(* IEC 61131-3 sources: TAuto/IEC 61131-3, 10 files *)

(* ---- FB_MB_PULL v.3.st ---- *)
FUNCTION_BLOCK MB_PULL

(* MB_PULL v.3 *)

(* MB_PULL - функциональный блок опроса по протоколу Modbus *)

(* Внешне задаются такие параметры как:
   - Команда выполнения/остановки цикла (ExecuteType);
   - Адрес/номер Slave-устройства (SlaveId);
   - Команда Modbus, которая реализована в FB MB_RTU_MASTER (Mode; 1, 2, 3, 4, 5, 6, 15, 16);
   - Начальный адрес регистров (Address);
   - Количество считываемых/записываемых данных (Count). *)
(* Внешне реализованы функции чтения/записи массива данных, в зависимости от  выбранной функции *)
(* Внутри функционального блока опроса используются следующие библиотечные функции:
   - MB_RTU_MASTER - функциональный блок Modbus;
   - MB_MASTER_QUEUE - структура созданная для команд Modbus. *)

// Первоначальная проверка, блок не выполняется
// MB_MS - экземпляр FB MB_RTU_MASTER
IF NOT MB_MS.Busy THEN                                                            // True - выполняется команда, False - не выполняется клманда

   QUEUE_INDEX := MB_Q.CurrentCommandIndex;                                       // Тип QUEUE_INDEX - INT. MB_Q - экземпляр MB_MASTER_QUEUE

   // Текущая команда завершилась
   IF MB_MS.Done THEN                                                             // Признак того, что команда завершилась

      // Текущий индекс команды
      MB_Q.CurrentCommandIndex := MB_Q.CurrentCommandIndex + 1;

      // Нет ошибок при выполнении FB
      IF MB_MS.Error = 0 THEN                                                     // 1. 0 - ошибок нет. 2. Диапазон 1..1000 - ошибки устройства Modbus. 3. Диапазон 1000..2000 - ошибки СПО. 4. Диапазон 2000+ - ошибки блока MB_RTU_MASTER

         // Задан корреткный режим выполнения
         IF  MB_Q.Commands[QUEUE_INDEX].ExecuteType <> 0 THEN

            // Сброс флага для режима "одиночного выполнения"
            IF MB_Q.Commands[QUEUE_INDEX].ExecuteType = 255 THEN

               MB_Q.Commands[QUEUE_INDEX].ExecuteType := 0;

            END_IF;

            (* Закомментированно потому что реализовано во внешних ST-программах *)

            // // Для операций чтения данных (1, 2, 3, 4 функции Modbus)
            // IF MB_Q.Commands[QUEUE_INDEX].Mode = 1                                // Чтение значений из нескольких регистров флагов - Read Coil Status
            //   OR MB_Q.Commands[QUEUE_INDEX].Mode = 2                              // Чтение значений из нескольких дискретных входов - Read Discrete Inputs
            //   OR MB_Q.Commands[QUEUE_INDEX].Mode = 3                              // Чтение значений из нескольких регистров хранения - Read Holding Registers
            //   OR MB_Q.Commands[QUEUE_INDEX].Mode = 4 THEN                         // Чтение значений из нескольких регистров ввода - Read Input Registers

            //   // Копирование данных полученных с устройства
            //   MB_Q.Commands[QUEUE_INDEX].Data := MB_MS.DataOut;                   // Массив считанных данных из Slave-устройства

            // END_IF;
         END_IF;
      END_IF;
   END_IF;

   // Сброс индекса запросов
   IF QUEUE_INDEX = 49 THEN

      MB_Q.CurrentCommandIndex := 0;

   END_IF;

   // Циклический перебор "карты памяти"
   FOR COMMAND_INDEX := MB_Q.CurrentCommandIndex TO 49 DO                            // Тип COMMAND_INDEX - INT

      // Сохранение текущего индекса
      MB_Q.CurrentCommandIndex := COMMAND_INDEX;

      // Задан корреткный режим выполнения
      IF MB_Q.Commands[COMMAND_INDEX].ExecuteType <> 0 THEN

         // Режим "выполнить один раз"
         IF MB_Q.Commands[COMMAND_INDEX].ExecuteType = 2 THEN

            MB_Q.Commands[COMMAND_INDEX].ExecuteType := 255;

         END_IF;

         (* Закомментированно потому что реализовано во внешних ST-программах *)

         // // Для операций записи данных (5, 6, 15, 16 функции Modbus)
         // IF  MB_Q.Commands[COMMAND_INDEX].Mode = 5                                   // Запись значения одного флага - Force Single Coil
         //    OR MB_Q.Commands[COMMAND_INDEX].Mode = 6                                 // Запись значения в один регистр хранения - Preset Single Register
         //    OR MB_Q.Commands[COMMAND_INDEX].Mode = 15                                // Запись значений в несколько регистров флагов - Force Multiple Coils
         //    OR MB_Q.Commands[COMMAND_INDEX].Mode = 16 THEN                           // Запись значений в несколько регистров хранения - Preset Multiple Registers

         //    // Копирование данных для записи в устройство
         //    MB_MS.DataIn := MB_Q.Commands[COMMAND_INDEX].Data;                       // Массив данных для записи в Slave-устройство

         // END_IF;

         // Настрока FB MB_RTU_MASTER
         MB_MS.Request := MB_REQUEST;                                                // Тип MB_REQUEST - BOOL. Команда выполнения/остановки опроса. Срабатывает по фронту, т.е. при смене входа с False на True
         MB_MS.SlaveId := MB_Q.Commands[COMMAND_INDEX].SlaveId;                      // Адрес/номер Slave-устройства
         MB_MS.Mode := MB_Q.Commands[COMMAND_INDEX].Mode;                            // Команда Modbus (1, 2, 3, 4, 5, 6, 15, 16)
         MB_MS.Address := MB_Q.Commands[COMMAND_INDEX].Address;                      // Начальный адрес register/coil (0 - 65535)
         MB_MS.Count := MB_Q.Commands[COMMAND_INDEX].Count;                          // Количество считываемых/записываемых данных. Зависит от типа данных register/coil (0 -123 для регистров , 0-246 для бит)

         EXIT;
      END_IF;
   END_FOR;
END_IF;

// Настройка параметров обмена FB MB_RTU_MASTER
MB_MS.BaudRate := MB_BaudRate;                                                       // Тип MB_BaudRate - UDINT. Скорость (9600, 19200, 38400, 57600, 115200 и др.)
MB_MS.Parity := MB_Parity;                                                           // Тип MB_Parity - BOOL. Бит чётности (True - есть контроль чётности)
MB_MS.StopBit := MB_StopBit;                                                         // Тип MB_StopBit - USINT. Количество стоповых бит (1, 2)
MB_MS.DataBit := MB_DataBit;                                                         // Тип MB_DataBit - USINT. Количество бит данных (7, 8)
MB_MS.TimeOut := MB_TimeOut;                                                         // Тип MB_TimeOut - UDINT. Время ожидания выполнения команды, мс
MB_MS.BusNumber := MB_BusNumber;                                                     // Тип MB_BusNumber - USINT. Локальная шина БЦП - 0,1; TCM/MI01 - 2-99
MB_MS.PortNumber := MB_PortNumber;                                                   // Тип MB_PortNumber - USINT. Номер порта/канала (0, 1. Если используется ТСМ, то значения: 0-7)
MB_MS();                                                                             // Вызов блока MB_RTUMASTER

// Вывод информации из блока MB_RTU_MASTER
// MB_DataOut := MB_MS.DataOut;                                                      // Тип MB_DataOut - USINT_0_245. Результаты выполнения опроса
MB_Busy := MB_MS.Busy;                                                            // Тип MB_Busy - BOOL. Выставляется в true если выполняется команда
MB_Done := MB_MS.Done;                                                            // Тип MB_Done - BOOL. Признак того, что команда завершилась
MB_Error := MB_MS.Error;                                                          // Тип MB_Error - UDINT. Ошибка
MB_ExecutionTime := MB_MS.ExecutionTime;                                          // Тип MB_ExecutionTime - UDINT. Время выполнения последней команды, мс
MB_AverageExecutionTime := MB_MS.AverageExecutionTime;                            // Тип MB_AverageExecutionTime - UDINT. Время выполнения последних четырёх команд, мс

// Сброс команды выполнения
// Закоментировать без вызова блока MB_RTUMASTER
IF MB_MS.Request THEN                                                             // Команда выполнения/остановки опроса. Срабатывает по фронту, т.е. при смене входа с False на True

   MB_MS.Request := False;                                                        // Остановка команды выполнения опроса

END_IF;

END_FUNCTION_BLOCK

(* ---- FB_MB_PULL v.4.st ---- *)
FUNCTION_BLOCK MB_PULL

(* MB_PULL v.3 *)

(* MB_PULL - функциональный блок опроса по протоколу Modbus *)

(* Внешне задаются такие параметры как:
   - Команда выполнения/остановки цикла (ExecuteType);
   - Адрес/номер Slave-устройства (SlaveId);
   - Команда Modbus, которая реализована в FB MB_RTU_MASTER (Mode; 1, 2, 3, 4, 5, 6, 15, 16);
   - Начальный адрес регистров (Address);
   - Количество считываемых/записываемых данных (Count). *)
(* Внешне реализованы функции чтения/записи массива данных, в зависимости от  выбранной функции *)
(* Внутри функционального блока опроса используются следующие библиотечные функции:
   - MB_RTU_MASTER - функциональный блок Modbus;
   - MB_MASTER_QUEUE - структура созданная для команд Modbus. *)

// Первоначальная проверка, блок не выполняется
// MB_MS - экземпляр FB MB_RTU_MASTER

HV_1185557(.Request, .SlaveId, .TimeOut, .Mode, .Address, .DataIn, .Count);
            BOOL       USINT     UDINT    USINT   UINT  USINT_0_245  UINT

  .DataOut, .Busy, .Done, .Error, .ExecutionTime, .AverageExecutionTime
 USINT_0_245  BOOL  BOOL   UDINT    UDINT             UDINT

MB_COM (ExecuteType, SlaveId, Mode, Address, Count)
        USINT           USINT  USINT UINT   UINT

MB_QUEUE(Commands, CurrentCommandIndex)
            [0..49]
        MB_COM_0_49        INT

IF NOT MB_MS.Busy THEN                                                            // True - выполняется команда, False - не выполняется клманда

   QUEUE_INDEX := MB_Q.CurrentCommandIndex;                                       // Тип QUEUE_INDEX - INT. MB_Q - экземпляр MB_MASTER_QUEUE

   // Текущая команда завершилась
   IF MB_MS.Done THEN                                                             // Признак того, что команда завершилась

      // Текущий индекс команды
      MB_Q.CurrentCommandIndex := MB_Q.CurrentCommandIndex + 1;

      // Нет ошибок при выполнении FB
      IF MB_MS.Error = 0 THEN                                                     // 1. 0 - ошибок нет. 2. Диапазон 1..1000 - ошибки устройства Modbus. 3. Диапазон 1000..2000 - ошибки СПО. 4. Диапазон 2000+ - ошибки блока MB_RTU_MASTER

         // Задан корреткный режим выполнения
         IF  MB_Q.Commands[QUEUE_INDEX].ExecuteType <> 0 THEN

            // Сброс флага для режима "одиночного выполнения"
            IF MB_Q.Commands[QUEUE_INDEX].ExecuteType = 255 THEN

               MB_Q.Commands[QUEUE_INDEX].ExecuteType := 0;

            END_IF;

            (* Закомментированно потому что реализовано во внешних ST-программах *)

            // // Для операций чтения данных (1, 2, 3, 4 функции Modbus)
            // IF MB_Q.Commands[QUEUE_INDEX].Mode = 1                                // Чтение значений из нескольких регистров флагов - Read Coil Status
            //   OR MB_Q.Commands[QUEUE_INDEX].Mode = 2                              // Чтение значений из нескольких дискретных входов - Read Discrete Inputs
            //   OR MB_Q.Commands[QUEUE_INDEX].Mode = 3                              // Чтение значений из нескольких регистров хранения - Read Holding Registers
            //   OR MB_Q.Commands[QUEUE_INDEX].Mode = 4 THEN                         // Чтение значений из нескольких регистров ввода - Read Input Registers

            //   // Копирование данных полученных с устройства
            //   MB_Q.Commands[QUEUE_INDEX].Data := MB_MS.DataOut;                   // Массив считанных данных из Slave-устройства

            // END_IF;
         END_IF;
      END_IF;
   END_IF;

   // Сброс индекса запросов
   IF QUEUE_INDEX = 49 THEN

      MB_Q.CurrentCommandIndex := 0;

   END_IF;

   // Циклический перебор "карты памяти"
   FOR COMMAND_INDEX := MB_Q.CurrentCommandIndex TO 49 DO                            // Тип COMMAND_INDEX - INT

      // Сохранение текущего индекса
      MB_Q.CurrentCommandIndex := COMMAND_INDEX;

      // Задан корреткный режим выполнения
      IF MB_Q.Commands[COMMAND_INDEX].ExecuteType <> 0 THEN

         // Режим "выполнить один раз"
         IF MB_Q.Commands[COMMAND_INDEX].ExecuteType = 2 THEN

            MB_Q.Commands[COMMAND_INDEX].ExecuteType := 255;

         END_IF;

         (* Закомментированно потому что реализовано во внешних ST-программах *)

         // // Для операций записи данных (5, 6, 15, 16 функции Modbus)
         // IF  MB_Q.Commands[COMMAND_INDEX].Mode = 5                                   // Запись значения одного флага - Force Single Coil
         //    OR MB_Q.Commands[COMMAND_INDEX].Mode = 6                                 // Запись значения в один регистр хранения - Preset Single Register
         //    OR MB_Q.Commands[COMMAND_INDEX].Mode = 15                                // Запись значений в несколько регистров флагов - Force Multiple Coils
         //    OR MB_Q.Commands[COMMAND_INDEX].Mode = 16 THEN                           // Запись значений в несколько регистров хранения - Preset Multiple Registers

         //    // Копирование данных для записи в устройство
         //    MB_MS.DataIn := MB_Q.Commands[COMMAND_INDEX].Data;                       // Массив данных для записи в Slave-устройство

         // END_IF;

         // Настрока FB MB_RTU_MASTER
         MB_MS.Request := MB_REQUEST;                                                // Тип MB_REQUEST - BOOL. Команда выполнения/остановки опроса. Срабатывает по фронту, т.е. при смене входа с False на True
         MB_MS.SlaveId := MB_Q.Commands[COMMAND_INDEX].SlaveId;                      // Адрес/номер Slave-устройства
         MB_MS.Mode := MB_Q.Commands[COMMAND_INDEX].Mode;                            // Команда Modbus (1, 2, 3, 4, 5, 6, 15, 16)
         MB_MS.Address := MB_Q.Commands[COMMAND_INDEX].Address;                      // Начальный адрес register/coil (0 - 65535)
         MB_MS.Count := MB_Q.Commands[COMMAND_INDEX].Count;                          // Количество считываемых/записываемых данных. Зависит от типа данных register/coil (0 -123 для регистров , 0-246 для бит)

         EXIT;
      END_IF;
   END_FOR;
END_IF;

// Настройка параметров обмена FB MB_RTU_MASTER
MB_MS.BaudRate := MB_BaudRate;                                                       // Тип MB_BaudRate - UDINT. Скорость (9600, 19200, 38400, 57600, 115200 и др.)
MB_MS.Parity := MB_Parity;                                                           // Тип MB_Parity - BOOL. Бит чётности (True - есть контроль чётности)
MB_MS.StopBit := MB_StopBit;                                                         // Тип MB_StopBit - USINT. Количество стоповых бит (1, 2)
MB_MS.DataBit := MB_DataBit;                                                         // Тип MB_DataBit - USINT. Количество бит данных (7, 8)
MB_MS.TimeOut := MB_TimeOut;                                                         // Тип MB_TimeOut - UDINT. Время ожидания выполнения команды, мс
MB_MS.BusNumber := MB_BusNumber;                                                     // Тип MB_BusNumber - USINT. Локальная шина БЦП - 0,1; TCM/MI01 - 2-99
MB_MS.PortNumber := MB_PortNumber;                                                   // Тип MB_PortNumber - USINT. Номер порта/канала (0, 1. Если используется ТСМ, то значения: 0-7)
MB_MS();                                                                             // Вызов блока MB_RTUMASTER

// Вывод информации из блока MB_RTU_MASTER
// MB_DataOut := MB_MS.DataOut;                                                      // Тип MB_DataOut - USINT_0_245. Результаты выполнения опроса
MB_Busy := MB_MS.Busy;                                                            // Тип MB_Busy - BOOL. Выставляется в true если выполняется команда
MB_Done := MB_MS.Done;                                                            // Тип MB_Done - BOOL. Признак того, что команда завершилась
MB_Error := MB_MS.Error;                                                          // Тип MB_Error - UDINT. Ошибка
MB_ExecutionTime := MB_MS.ExecutionTime;                                          // Тип MB_ExecutionTime - UDINT. Время выполнения последней команды, мс
MB_AverageExecutionTime := MB_MS.AverageExecutionTime;                            // Тип MB_AverageExecutionTime - UDINT. Время выполнения последних четырёх команд, мс

// Сброс команды выполнения
// Закоментировать без вызова блока MB_RTUMASTER
IF MB_MS.Request THEN                                                             // Команда выполнения/остановки опроса. Срабатывает по фронту, т.е. при смене входа с False на True

   MB_MS.Request := False;                                                        // Остановка команды выполнения опроса

END_IF;

END_FUNCTION_BLOCK

(* ---- FUNCTION_BLOCK MB_PULL.st ---- *)
FUNCTION_BLOCK MB_PULL

(* MB_PULL v.3 *)

(* MB_PULL - функциональный блок опроса по протоколу Modbus *)

(* Внешне задаются такие параметры как:
   - Команда выполнения/остановки цикла (ExecuteType);
   - Адрес/номер Slave-устройства (SlaveId);
   - Команда Modbus, которая реализована в FB MB_RTU_MASTER (Mode; 1, 2, 3, 4, 5, 6, 15, 16);
   - Начальный адрес регистров (Address);
   - Количество считываемых/записываемых данных (Count). *)
(* Внешне реализованы функции чтения/записи массива данных, в зависимости от  выбранной функции *)
(* Внутри функционального блока опроса используются следующие библиотечные функции:
   - MB_RTU_MASTER - функциональный блок Modbus;
   - MB_MASTER_QUEUE - структура созданная для команд Modbus. *)

// Первоначальная проверка, блок не выполняется
// MB_MS - экземпляр FB MB_RTU_MASTER
IF NOT MB_MS.Busy THEN                                                            // True - выполняется команда, False - не выполняется клманда

    // Текущая команда завершилась
    IF MB_MS.Done THEN                                                             // Признак того, что команда завершилась

    // Текущий индекс команды
    MB_Q.CurrentCommandIndex := MB_Q.CurrentCommandIndex + 1;

        // Нет ошибок при выполнении FB
        IF MB_MS.Error = 0 THEN                                                     // 1. 0 - ошибок нет. 2. Диапазон 1..1000 - ошибки устройства Modbus. 3. Диапазон 1000..2000 - ошибки СПО. 4. Диапазон 2000+ - ошибки блока MB_RTU_MASTER

CASE MB_Q.CurrentCommandIndex OF
1:
QUEUE_INDEX := 1;
2:
QUEUE_INDEX := 2;
3:
QUEUE_INDEX := 3;
4:
QUEUE_INDEX := 4;
5:
QUEUE_INDEX := 5;
6:
QUEUE_INDEX := 6;
7:
QUEUE_INDEX := 7;
8:
QUEUE_INDEX := 8;
9:
QUEUE_INDEX := 9;
10:
QUEUE_INDEX := 10;
MB_Q.CurrentCommandIndex := 0;
END_CASE;

         // Задан корреткный режим выполнения
         IF  MB_Q.Commands[QUEUE_INDEX].ExecuteType <> 0 THEN

            // Сброс флага для режима "одиночного выполнения"
            IF MB_Q.Commands[QUEUE_INDEX].ExecuteType = 255 THEN

               MB_Q.Commands[QUEUE_INDEX].ExecuteType := 0;

            END_IF;

                    END_IF;
      END_IF;
   END_IF;

   // Сброс индекса запросов
   IF QUEUE_INDEX = 49 THEN

      MB_Q.CurrentCommandIndex := 0;

   END_IF;

   // Циклический перебор "карты памяти"
   FOR COMMAND_INDEX := MB_Q.CurrentCommandIndex TO 49 DO                            // Тип COMMAND_INDEX - INT

      // Сохранение текущего индекса
      MB_Q.CurrentCommandIndex := COMMAND_INDEX;

      // Задан корреткный режим выполнения
      IF MB_Q.Commands[COMMAND_INDEX].ExecuteType <> 0 THEN

         // Режим "выполнить один раз"
         IF MB_Q.Commands[COMMAND_INDEX].ExecuteType = 2 THEN

            MB_Q.Commands[COMMAND_INDEX].ExecuteType := 255;

         END_IF;

         (* Закомментированно потому что реализовано во внешних ST-программах *)

         // // Для операций записи данных (5, 6, 15, 16 функции Modbus)
         // IF  MB_Q.Commands[COMMAND_INDEX].Mode = 5                                   // Запись значения одного флага - Force Single Coil
         //    OR MB_Q.Commands[COMMAND_INDEX].Mode = 6                                 // Запись значения в один регистр хранения - Preset Single Register
         //    OR MB_Q.Commands[COMMAND_INDEX].Mode = 15                                // Запись значений в несколько регистров флагов - Force Multiple Coils
         //    OR MB_Q.Commands[COMMAND_INDEX].Mode = 16 THEN                           // Запись значений в несколько регистров хранения - Preset Multiple Registers

         //    // Копирование данных для записи в устройство
         //    MB_MS.DataIn := MB_Q.Commands[COMMAND_INDEX].Data;                       // Массив данных для записи в Slave-устройство

         // END_IF;

         // Настрока FB MB_RTU_MASTER
         MB_MS.Request := MB_REQUEST;                                                // Тип MB_REQUEST - BOOL. Команда выполнения/остановки опроса. Срабатывает по фронту, т.е. при смене входа с False на True
         MB_MS.SlaveId := MB_Q.Commands[COMMAND_INDEX].SlaveId;                      // Адрес/номер Slave-устройства
         MB_MS.Mode := MB_Q.Commands[COMMAND_INDEX].Mode;                            // Команда Modbus (1, 2, 3, 4, 5, 6, 15, 16)
         MB_MS.Address := MB_Q.Commands[COMMAND_INDEX].Address;                      // Начальный адрес register/coil (0 - 65535)
         MB_MS.Count := MB_Q.Commands[COMMAND_INDEX].Count;                          // Количество считываемых/записываемых данных. Зависит от типа данных register/coil (0 -123 для регистров , 0-246 для бит)

         EXIT;
      END_IF;
   END_FOR;
END_IF;

// Настройка параметров обмена FB MB_RTU_MASTER
MB_MS.BaudRate := MB_BaudRate;                                                       // Тип MB_BaudRate - UDINT. Скорость (9600, 19200, 38400, 57600, 115200 и др.)
MB_MS.Parity := MB_Parity;                                                           // Тип MB_Parity - BOOL. Бит чётности (True - есть контроль чётности)
MB_MS.StopBit := MB_StopBit;                                                         // Тип MB_StopBit - USINT. Количество стоповых бит (1, 2)
MB_MS.DataBit := MB_DataBit;                                                         // Тип MB_DataBit - USINT. Количество бит данных (7, 8)
MB_MS.TimeOut := MB_TimeOut;                                                         // Тип MB_TimeOut - UDINT. Время ожидания выполнения команды, мс
MB_MS.BusNumber := MB_BusNumber;                                                     // Тип MB_BusNumber - USINT. Локальная шина БЦП - 0,1; TCM/MI01 - 2-99
MB_MS.PortNumber := MB_PortNumber;                                                   // Тип MB_PortNumber - USINT. Номер порта/канала (0, 1. Если используется ТСМ, то значения: 0-7)
MB_MS();                                                                             // Вызов блока MB_RTUMASTER

// Вывод информации из блока MB_RTU_MASTER
// MB_DataOut := MB_MS.DataOut;                                                      // Тип MB_DataOut - USINT_0_245. Результаты выполнения опроса
MB_Busy := MB_MS.Busy;                                                            // Тип MB_Busy - BOOL. Выставляется в true если выполняется команда
MB_Done := MB_MS.Done;                                                            // Тип MB_Done - BOOL. Признак того, что команда завершилась
MB_Error := MB_MS.Error;                                                          // Тип MB_Error - UDINT. Ошибка
MB_ExecutionTime := MB_MS.ExecutionTime;                                          // Тип MB_ExecutionTime - UDINT. Время выполнения последней команды, мс
MB_AverageExecutionTime := MB_MS.AverageExecutionTime;                            // Тип MB_AverageExecutionTime - UDINT. Время выполнения последних четырёх команд, мс

// Сброс команды выполнения
// Закоментировать без вызова блока MB_RTUMASTER
IF MB_MS.Request THEN                                                             // Команда выполнения/остановки опроса. Срабатывает по фронту, т.е. при смене входа с False на True

   MB_MS.Request := False;                                                        // Остановка команды выполнения опроса

END_IF;

END_FUNCTION_BLOCK

(* ---- IO_control.st ---- *)
PROGRAM IO_control

(***************************************************************************)
// ЛОКАЛЬНАЯ ШИНА 0
(***************************************************************************)

// [2] DO32
_IO_Q1_DO32_0_VAL.Measurement := UB_0_0_DO32_CH0_OUT;
_IO_Q1_DO32_1_VAL.Measurement := UB_0_0_DO32_CH1_OUT;
_IO_Q1_DO32_2_VAL.Measurement := UB_0_0_DO32_CH2_OUT;
_IO_Q1_DO32_3_VAL.Measurement := UB_0_0_DO32_CH3_OUT;
_IO_Q1_DO32_4_VAL.Measurement := UB_0_0_DO32_CH4_OUT;
_IO_Q1_DO32_5_VAL.Measurement := UB_0_0_DO32_CH5_OUT;
_IO_Q1_DO32_6_VAL.Measurement := UB_0_0_DO32_CH6_OUT;
_IO_Q1_DO32_7_VAL.Measurement := UB_0_0_DO32_CH7_OUT;
_IO_Q1_DO32_8_VAL.Measurement := UB_0_0_DO32_CH8_OUT;
_IO_Q1_DO32_9_VAL.Measurement := UB_0_0_DO32_CH9_OUT;
_IO_Q1_DO32_10_VAL.Measurement := UB_0_0_DO32_CH10_OUT;
_IO_Q1_DO32_11_VAL.Measurement := UB_0_0_DO32_CH11_OUT;
_IO_Q1_DO32_12_VAL.Measurement := UB_0_0_DO32_CH12_OUT;
_IO_Q1_DO32_13_VAL.Measurement := UB_0_0_DO32_CH13_OUT;
_IO_Q1_DO32_14_VAL.Measurement := UB_0_0_DO32_CH14_OUT;
_IO_Q1_DO32_15_VAL.Measurement := UB_0_0_DO32_CH15_OUT;
_IO_Q1_DO32_16_VAL.Measurement := UB_0_0_DO32_CH16_OUT;
_IO_Q1_DO32_17_VAL.Measurement := UB_0_0_DO32_CH17_OUT;
_IO_Q1_DO32_18_VAL.Measurement := UB_0_0_DO32_CH18_OUT;
_IO_Q1_DO32_19_VAL.Measurement := UB_0_0_DO32_CH19_OUT;
_IO_Q1_DO32_20_VAL.Measurement := UB_0_0_DO32_CH20_OUT;
_IO_Q1_DO32_21_VAL.Measurement := UB_0_0_DO32_CH21_OUT;
_IO_Q1_DO32_22_VAL.Measurement := UB_0_0_DO32_CH22_OUT;
_IO_Q1_DO32_23_VAL.Measurement := UB_0_0_DO32_CH23_OUT;
_IO_Q1_DO32_24_VAL.Measurement := UB_0_0_DO32_CH24_OUT;
_IO_Q1_DO32_25_VAL.Measurement := UB_0_0_DO32_CH25_OUT;
_IO_Q1_DO32_26_VAL.Measurement := UB_0_0_DO32_CH26_OUT;
_IO_Q1_DO32_27_VAL.Measurement := UB_0_0_DO32_CH27_OUT;
_IO_Q1_DO32_28_VAL.Measurement := UB_0_0_DO32_CH28_OUT;
_IO_Q1_DO32_29_VAL.Measurement := UB_0_0_DO32_CH29_OUT;
_IO_Q1_DO32_30_VAL.Measurement := UB_0_0_DO32_CH30_OUT;
_IO_Q1_DO32_31_VAL.Measurement := UB_0_0_DO32_CH31_OUT;

END_PROGRAM

(* ---- IO_RT.st ---- *)
PROGRAM IO_RT

//ВЫЗОВ ГЕНЕРАТОРОВ
GENERATOR(.StartGener, .PulseTime, .ResetCnt);
SIG_GEN_1(.RUN, .PERIOD, .MAXIMUM);

// НАСТРОЙКА ФБ AD
AD_VALID_DOWN := -100000;
AD_VALID_UP := 100000;
AD_IN0 := 10;
AD_IN100 := 100;

// КВИТИРОВАНИЕ
TIMER_REAL(FALSE, 0, 0, 10, T#20ms);

TMB_1_0_DI32_KVIT := TIMER_REAL.Out;
TMB_1_0_DO32_KVIT := TIMER_REAL.Out;
TMB_1_0_AIG16_KVIT := TIMER_REAL.Out;
TMB_1_0_AI8_KVIT := TIMER_REAL.Out;
TMB_1_0_AOC4_KVIT := TIMER_REAL.Out;

// ИНТЕГРАЛЬНЫЙ ПОАЗАТЕЛЬ ШИНЫ
IF TMB_1_0_DI32_INTEGRAL_VAL_QUALITY AND
    TMB_1_0_DO32_INTEGRAL_VAL_DIAG_QUALITY AND
    TMB_1_0_AIG16_INTEGRAL_VAL_QUALITY AND
    TMB_1_0_AI8_INTEGRAL_VAL_QUALITY AND
    TMB_1_0_AOC4_INTEGRAL_VAL_DIAG_QUALITY

    THEN TMB_1_0_TMB_QUALITY := TRUE;
    ELSE TMB_1_0_TMB_QUALITY := FALSE;
END_IF;

END_PROGRAM

(* ---- IO_SF.st ---- *)
PROGRAM IO

//ВЫЗОВ ГЕНЕРАТОРОВ
GENERATOR(.StartGener, .PulseTime, .ResetCnt);
SIG_GEN_1(.RUN, .PERIOD, .MAXIMUM);

// НАСТРОЙКА ФБ AD
AD_VALID_DOWN := -100000;
AD_VALID_UP := 100000;
AD_IN0 := 10;
AD_IN100 := 100;

// КВИТИРОВАНИЕ
TIMER_REAL(FALSE, 0, 0, 10, T#20ms);

UB_0_0_DI32_KVIT := TIMER_REAL.Out;
UB_0_0_DO32_KVIT := TIMER_REAL.Out;
UB_0_0_AIG16_KVIT := TIMER_REAL.Out;
UB_0_0_AI8_KVIT := TIMER_REAL.Out;
UB_0_0_AOC4_KVIT := TIMER_REAL.Out;

UB_0_32_DI32_KVIT := TIMER_REAL.Out;
UB_0_32_DO32_KVIT := TIMER_REAL.Out;
UB_0_32_AIG16_KVIT := TIMER_REAL.Out;
UB_0_32_AI8_KVIT := TIMER_REAL.Out;
UB_0_32_AOC4_KVIT := TIMER_REAL.Out;

UB_1_0_DI32_KVIT := TIMER_REAL.Out;
UB_1_0_DO32_KVIT := TIMER_REAL.Out;
UB_1_0_AIG16_KVIT := TIMER_REAL.Out;
UB_1_0_AI8_KVIT := TIMER_REAL.Out;
UB_1_0_AOC4_KVIT := TIMER_REAL.Out;

UB_12_0_DI32_KVIT := TIMER_REAL.Out;
UB_12_0_DO32_KVIT := TIMER_REAL.Out;
UB_12_0_AIG16_KVIT := TIMER_REAL.Out;
UB_12_0_AI8_KVIT := TIMER_REAL.Out;
UB_12_0_AOC4_KVIT := TIMER_REAL.Out;

UB_22_0_DI32_KVIT := TIMER_REAL.Out;
UB_22_0_DO32_KVIT := TIMER_REAL.Out;
UB_22_0_AIG16_KVIT := TIMER_REAL.Out;
UB_22_0_AI8_KVIT := TIMER_REAL.Out;
UB_22_0_AOC4_KVIT := TIMER_REAL.Out;

// ИНТЕГРАЛЬНЫЙ ПОАЗАТЕЛЬ ШИНЫ
IF UB_0_0_DI32_INTEGRAL_VAL_QUALITY AND
    UB_0_0_DO32_INTEGRAL_VAL_DIAG_QUALITY AND
    UB_0_0_AIG16_INTEGRAL_VAL_QUALITY AND
    UB_0_0_AI8_INTEGRAL_VAL_QUALITY AND
    UB_0_0_AOC4_INTEGRAL_VAL_DIAG_QUALITY

    THEN UB_0_0_UNITBAS_QUALITY := TRUE;
    ELSE UB_0_0_UNITBAS_QUALITY := FALSE;
END_IF;

IF UB_0_32_DI32_INTEGRAL_VAL_QUALITY AND
    UB_0_32_DO32_INTEGRAL_VAL_DIAG_QUALITY AND
    UB_0_32_AIG16_INTEGRAL_VAL_QUALITY AND
    UB_0_32_AI8_INTEGRAL_VAL_QUALITY AND
    UB_0_32_AOC4_INTEGRAL_VAL_DIAG_QUALITY

    THEN UB_0_32_UNITBAS_QUALITY := TRUE;
    ELSE UB_0_32_UNITBAS_QUALITY := FALSE;
END_IF;

IF UB_1_0_DI32_INTEGRAL_VAL_QUALITY AND
    UB_1_0_DO32_INTEGRAL_VAL_DIAG_QUALITY AND
    UB_1_0_AIG16_INTEGRAL_VAL_QUALITY AND
    UB_1_0_AI8_INTEGRAL_VAL_QUALITY AND
    UB_1_0_AOC4_INTEGRAL_VAL_DIAG_QUALITY

    THEN UB_1_0_UNITBAS_QUALITY := TRUE;
    ELSE UB_1_0_UNITBAS_QUALITY := FALSE;
END_IF;

IF UB_12_0_DI32_INTEGRAL_VAL_QUALITY AND
    UB_12_0_DO32_INTEGRAL_VAL_DIAG_QUALITY AND
    UB_12_0_AIG16_INTEGRAL_VAL_QUALITY AND
    UB_12_0_AI8_INTEGRAL_VAL_QUALITY AND
    UB_12_0_AOC4_INTEGRAL_VAL_DIAG_QUALITY

    THEN UB_12_0_UNITBAS_QUALITY := TRUE;
    ELSE UB_12_0_UNITBAS_QUALITY := FALSE;
END_IF;

IF UB_22_0_DI32_INTEGRAL_VAL_QUALITY AND
    UB_22_0_DO32_INTEGRAL_VAL_DIAG_QUALITY AND
    UB_22_0_AIG16_INTEGRAL_VAL_QUALITY AND
    UB_22_0_AI8_INTEGRAL_VAL_QUALITY AND
    UB_22_0_AOC4_INTEGRAL_VAL_DIAG_QUALITY

    THEN UB_22_0_UNITBAS_QUALITY := TRUE;
    ELSE UB_22_0_UNITBAS_QUALITY := FALSE;
END_IF;

END_PROGRAM

(* ---- PRG CPU715_Modbus.st ---- *)
PROGRAM CPU715_Modbus

(* Программа для передачи данных по протоколу Modbus *)

(* Генерация осуществляется с помощью ФБ MultiTypeGener *)
(* Диапазон регистров:
        для IR, HR:
            DINT - 32000...41999
            REAL - 42000...51999
            INT - 52000...61999
        для CL, DI:
            BOOL - 32000...41999 *)
(* Используемые каналы 0-97 для каждого типа данных *)

(* Считывание CL регистров *)
    // Переменные BOOL, регистры - 32000...41999
        _IO_QX5_1_0 := RESVAR_BOOL;
        _IO_QX5_1_1 := RESVAR_BOOL;
        _IO_QX5_1_2 := RESVAR_BOOL;
        _IO_QX5_1_3 := RESVAR_BOOL;
        _IO_QX5_1_4 := RESVAR_BOOL;
        _IO_QX5_1_5 := RESVAR_BOOL;
        _IO_QX5_1_6 := RESVAR_BOOL;
        _IO_QX5_1_7 := RESVAR_BOOL;
        _IO_QX5_1_8 := RESVAR_BOOL;
        _IO_QX5_1_9 := RESVAR_BOOL;
        _IO_QX5_1_10 := RESVAR_BOOL;
        _IO_QX5_1_11 := RESVAR_BOOL;
        _IO_QX5_1_12 := RESVAR_BOOL;
        _IO_QX5_1_13 := RESVAR_BOOL;

        _IO_QX5_1_14 := RESVAR_BOOL;
        _IO_QX5_1_15 := RESVAR_BOOL;
        _IO_QX5_1_16 := RESVAR_BOOL;
        _IO_QX5_1_17 := RESVAR_BOOL;
        _IO_QX5_1_18 := RESVAR_BOOL;
        _IO_QX5_1_19 := RESVAR_BOOL;
        _IO_QX5_1_20 := RESVAR_BOOL;
        _IO_QX5_1_21 := RESVAR_BOOL;
        _IO_QX5_1_22 := RESVAR_BOOL;
        _IO_QX5_1_23 := RESVAR_BOOL;
        _IO_QX5_1_24 := RESVAR_BOOL;
        _IO_QX5_1_25 := RESVAR_BOOL;
        _IO_QX5_1_26 := RESVAR_BOOL;
        _IO_QX5_1_27 := RESVAR_BOOL;

        _IO_QX5_1_28 := RESVAR_BOOL;
        _IO_QX5_1_29 := RESVAR_BOOL;
        _IO_QX5_1_30 := RESVAR_BOOL;
        _IO_QX5_1_31 := RESVAR_BOOL;
        _IO_QX5_1_32 := RESVAR_BOOL;
        _IO_QX5_1_33 := RESVAR_BOOL;
        _IO_QX5_1_34 := RESVAR_BOOL;
        _IO_QX5_1_35 := RESVAR_BOOL;
        _IO_QX5_1_36 := RESVAR_BOOL;
        _IO_QX5_1_37 := RESVAR_BOOL;
        _IO_QX5_1_38 := RESVAR_BOOL;
        _IO_QX5_1_39 := RESVAR_BOOL;
        _IO_QX5_1_40 := RESVAR_BOOL;
        _IO_QX5_1_41 := RESVAR_BOOL;

        _IO_QX5_1_42 := RESVAR_BOOL;
        _IO_QX5_1_43 := RESVAR_BOOL;
        _IO_QX5_1_44 := RESVAR_BOOL;
        _IO_QX5_1_45 := RESVAR_BOOL;
        _IO_QX5_1_46 := RESVAR_BOOL;
        _IO_QX5_1_47 := RESVAR_BOOL;
        _IO_QX5_1_48 := RESVAR_BOOL;
        _IO_QX5_1_49 := RESVAR_BOOL;
        _IO_QX5_1_50 := RESVAR_BOOL;
        _IO_QX5_1_51 := RESVAR_BOOL;
        _IO_QX5_1_52 := RESVAR_BOOL;
        _IO_QX5_1_53 := RESVAR_BOOL;
        _IO_QX5_1_54 := RESVAR_BOOL;
        _IO_QX5_1_55 := RESVAR_BOOL;

        _IO_QX5_1_56 := RESVAR_BOOL;
        _IO_QX5_1_57 := RESVAR_BOOL;
        _IO_QX5_1_58 := RESVAR_BOOL;
        _IO_QX5_1_59 := RESVAR_BOOL;
        _IO_QX5_1_60 := RESVAR_BOOL;
        _IO_QX5_1_61 := RESVAR_BOOL;
        _IO_QX5_1_62 := RESVAR_BOOL;
        _IO_QX5_1_63 := RESVAR_BOOL;
        _IO_QX5_1_64 := RESVAR_BOOL;
        _IO_QX5_1_65 := RESVAR_BOOL;
        _IO_QX5_1_66 := RESVAR_BOOL;
        _IO_QX5_1_67 := RESVAR_BOOL;
        _IO_QX5_1_68 := RESVAR_BOOL;
        _IO_QX5_1_69 := RESVAR_BOOL;

        _IO_QX5_1_70 := RESVAR_BOOL;
        _IO_QX5_1_71 := RESVAR_BOOL;
        _IO_QX5_1_72 := RESVAR_BOOL;
        _IO_QX5_1_73 := RESVAR_BOOL;
        _IO_QX5_1_74 := RESVAR_BOOL;
        _IO_QX5_1_75 := RESVAR_BOOL;
        _IO_QX5_1_76 := RESVAR_BOOL;
        _IO_QX5_1_77 := RESVAR_BOOL;
        _IO_QX5_1_78 := RESVAR_BOOL;
        _IO_QX5_1_79 := RESVAR_BOOL;
        _IO_QX5_1_80 := RESVAR_BOOL;
        _IO_QX5_1_81 := RESVAR_BOOL;
        _IO_QX5_1_82 := RESVAR_BOOL;
        _IO_QX5_1_83 := RESVAR_BOOL;

        _IO_QX5_1_84 := RESVAR_BOOL;
        _IO_QX5_1_85 := RESVAR_BOOL;
        _IO_QX5_1_86 := RESVAR_BOOL;
        _IO_QX5_1_87 := RESVAR_BOOL;
        _IO_QX5_1_88 := RESVAR_BOOL;
        _IO_QX5_1_89 := RESVAR_BOOL;
        _IO_QX5_1_90 := RESVAR_BOOL;
        _IO_QX5_1_91 := RESVAR_BOOL;
        _IO_QX5_1_92 := RESVAR_BOOL;
        _IO_QX5_1_93 := RESVAR_BOOL;
        _IO_QX5_1_94 := RESVAR_BOOL;
        _IO_QX5_1_95 := RESVAR_BOOL;
        _IO_QX5_1_96 := RESVAR_BOOL;
        _IO_QX5_1_97 := RESVAR_BOOL;

(* Считывание DI регистров *)
    // Переменные BOOL, регистры - 32000...41999
        _IO_QU7_0 := RESVAR_BOOL;
        _IO_QU7_1 := RESVAR_BOOL;
        _IO_QU7_2 := RESVAR_BOOL;
        _IO_QU7_3 := RESVAR_BOOL;
        _IO_QU7_4 := RESVAR_BOOL;
        _IO_QU7_5 := RESVAR_BOOL;
        _IO_QU7_6 := RESVAR_BOOL;
        _IO_QU7_7 := RESVAR_BOOL;
        _IO_QU7_8 := RESVAR_BOOL;
        _IO_QU7_9 := RESVAR_BOOL;
        _IO_QU7_10 := RESVAR_BOOL;
        _IO_QU7_11 := RESVAR_BOOL;
        _IO_QU7_12 := RESVAR_BOOL;
        _IO_QU7_13 := RESVAR_BOOL;

        _IO_QU7_14 := RESVAR_BOOL;
        _IO_QU7_15 := RESVAR_BOOL;
        _IO_QU7_16 := RESVAR_BOOL;
        _IO_QU7_17 := RESVAR_BOOL;
        _IO_QU7_18 := RESVAR_BOOL;
        _IO_QU7_19 := RESVAR_BOOL;
        _IO_QU7_20 := RESVAR_BOOL;
        _IO_QU7_21 := RESVAR_BOOL;
        _IO_QU7_22 := RESVAR_BOOL;
        _IO_QU7_23 := RESVAR_BOOL;
        _IO_QU7_24 := RESVAR_BOOL;
        _IO_QU7_25 := RESVAR_BOOL;
        _IO_QU7_26 := RESVAR_BOOL;
        _IO_QU7_27 := RESVAR_BOOL;

        _IO_QU7_28 := RESVAR_BOOL;
        _IO_QU7_29 := RESVAR_BOOL;
        _IO_QU7_30 := RESVAR_BOOL;
        _IO_QU7_31 := RESVAR_BOOL;
        _IO_QU7_32 := RESVAR_BOOL;
        _IO_QU7_33 := RESVAR_BOOL;
        _IO_QU7_34 := RESVAR_BOOL;
        _IO_QU7_35 := RESVAR_BOOL;
        _IO_QU7_36 := RESVAR_BOOL;
        _IO_QU7_37 := RESVAR_BOOL;
        _IO_QU7_38 := RESVAR_BOOL;
        _IO_QU7_39 := RESVAR_BOOL;
        _IO_QU7_40 := RESVAR_BOOL;
        _IO_QU7_41 := RESVAR_BOOL;

        _IO_QU7_42 := RESVAR_BOOL;
        _IO_QU7_43 := RESVAR_BOOL;
        _IO_QU7_44 := RESVAR_BOOL;
        _IO_QU7_45 := RESVAR_BOOL;
        _IO_QU7_46 := RESVAR_BOOL;
        _IO_QU7_47 := RESVAR_BOOL;
        _IO_QU7_48 := RESVAR_BOOL;
        _IO_QU7_49 := RESVAR_BOOL;
        _IO_QU7_50 := RESVAR_BOOL;
        _IO_QU7_51 := RESVAR_BOOL;
        _IO_QU7_52 := RESVAR_BOOL;
        _IO_QU7_53 := RESVAR_BOOL;
        _IO_QU7_54 := RESVAR_BOOL;
        _IO_QU7_55 := RESVAR_BOOL;

        _IO_QU7_56 := RESVAR_BOOL;
        _IO_QU7_57 := RESVAR_BOOL;
        _IO_QU7_58 := RESVAR_BOOL;
        _IO_QU7_59 := RESVAR_BOOL;
        _IO_QU7_60 := RESVAR_BOOL;
        _IO_QU7_61 := RESVAR_BOOL;
        _IO_QU7_62 := RESVAR_BOOL;
        _IO_QU7_63 := RESVAR_BOOL;
        _IO_QU7_64 := RESVAR_BOOL;
        _IO_QU7_65 := RESVAR_BOOL;
        _IO_QU7_66 := RESVAR_BOOL;
        _IO_QU7_67 := RESVAR_BOOL;
        _IO_QU7_68 := RESVAR_BOOL;
        _IO_QU7_69 := RESVAR_BOOL;

        _IO_QU7_70 := RESVAR_BOOL;
        _IO_QU7_71 := RESVAR_BOOL;
        _IO_QU7_72 := RESVAR_BOOL;
        _IO_QU7_73 := RESVAR_BOOL;
        _IO_QU7_74 := RESVAR_BOOL;
        _IO_QU7_75 := RESVAR_BOOL;
        _IO_QU7_76 := RESVAR_BOOL;
        _IO_QU7_77 := RESVAR_BOOL;
        _IO_QU7_78 := RESVAR_BOOL;
        _IO_QU7_79 := RESVAR_BOOL;
        _IO_QU7_80 := RESVAR_BOOL;
        _IO_QU7_81 := RESVAR_BOOL;
        _IO_QU7_82 := RESVAR_BOOL;
        _IO_QU7_83 := RESVAR_BOOL;

        _IO_QU7_84 := RESVAR_BOOL;
        _IO_QU7_85 := RESVAR_BOOL;
        _IO_QU7_86 := RESVAR_BOOL;
        _IO_QU7_87 := RESVAR_BOOL;
        _IO_QU7_88 := RESVAR_BOOL;
        _IO_QU7_89 := RESVAR_BOOL;
        _IO_QU7_90 := RESVAR_BOOL;
        _IO_QU7_91 := RESVAR_BOOL;
        _IO_QU7_92 := RESVAR_BOOL;
        _IO_QU7_93 := RESVAR_BOOL;
        _IO_QU7_94 := RESVAR_BOOL;
        _IO_QU7_95 := RESVAR_BOOL;
        _IO_QU7_96 := RESVAR_BOOL;
        _IO_QU7_97 := RESVAR_BOOL;

(* Считывание HR регистров *)
    // Переменные DINT, регистры - 32000...41999
        _IO_QX0_1_0 := ANY_TO_DINT(RESVAR_BYTE);
        _IO_QX0_1_1 := ANY_TO_DINT(RESVAR_WORD);
        _IO_QX0_1_2 := RESVAR_DWORD;
        _IO_QX0_1_3 := ANY_TO_DINT(RESVAR_LWORD);
        _IO_QX0_1_4 := ANY_TO_DINT(RESVAR_SINT);
        _IO_QX0_1_5 := ANY_TO_DINT(RESVAR_INT);
        _IO_QX0_1_6 := RESVAR_DINT;
        _IO_QX0_1_7 := ANY_TO_DINT(RESVAR_LINT);
        _IO_QX0_1_8 := ANY_TO_DINT(RESVAR_USINT);
        _IO_QX0_1_9 := ANY_TO_DINT(RESVAR_UINT);
        _IO_QX0_1_10 := RESVAR_UDINT;
        _IO_QX0_1_11 := ANY_TO_DINT(RESVAR_ULINT);
        _IO_QX0_1_12 := ANY_TO_DINT(RESVAR_REAL);
        _IO_QX0_1_13 := ANY_TO_DINT(RESVAR_LREAL);

        _IO_QX0_1_14 := ANY_TO_DINT(RESVAR_BYTE);
        _IO_QX0_1_15 := ANY_TO_DINT(RESVAR_WORD);
        _IO_QX0_1_16 := RESVAR_DWORD;
        _IO_QX0_1_17 := ANY_TO_DINT(RESVAR_LWORD);
        _IO_QX0_1_18 := ANY_TO_DINT(RESVAR_SINT);
        _IO_QX0_1_19 := ANY_TO_DINT(RESVAR_INT);
        _IO_QX0_1_20 := RESVAR_DINT;
        _IO_QX0_1_21 := ANY_TO_DINT(RESVAR_LINT);
        _IO_QX0_1_22 := ANY_TO_DINT(RESVAR_USINT);
        _IO_QX0_1_23 := ANY_TO_DINT(RESVAR_UINT);
        _IO_QX0_1_24 := RESVAR_UDINT;
        _IO_QX0_1_25 := ANY_TO_DINT(RESVAR_ULINT);
        _IO_QX0_1_26 := ANY_TO_DINT(RESVAR_REAL);
        _IO_QX0_1_27 := ANY_TO_DINT(RESVAR_LREAL);

        _IO_QX0_1_28 := ANY_TO_DINT(RESVAR_BYTE);
        _IO_QX0_1_29 := ANY_TO_DINT(RESVAR_WORD);
        _IO_QX0_1_30 := RESVAR_DWORD;
        _IO_QX0_1_31 := ANY_TO_DINT(RESVAR_LWORD);
        _IO_QX0_1_32 := ANY_TO_DINT(RESVAR_SINT);
        _IO_QX0_1_33 := ANY_TO_DINT(RESVAR_INT);
        _IO_QX0_1_34 := RESVAR_DINT;
        _IO_QX0_1_35 := ANY_TO_DINT(RESVAR_LINT);
        _IO_QX0_1_36 := ANY_TO_DINT(RESVAR_USINT);
        _IO_QX0_1_37 := ANY_TO_DINT(RESVAR_UINT);
        _IO_QX0_1_38 := RESVAR_UDINT;
        _IO_QX0_1_39 := ANY_TO_DINT(RESVAR_ULINT);
        _IO_QX0_1_40 := ANY_TO_DINT(RESVAR_REAL);
        _IO_QX0_1_41 := ANY_TO_DINT(RESVAR_LREAL);

        _IO_QX0_1_42 := ANY_TO_DINT(RESVAR_BYTE);
        _IO_QX0_1_43 := ANY_TO_DINT(RESVAR_WORD);
        _IO_QX0_1_44 := RESVAR_DWORD;
        _IO_QX0_1_45 := ANY_TO_DINT(RESVAR_LWORD);
        _IO_QX0_1_46 := ANY_TO_DINT(RESVAR_SINT);
        _IO_QX0_1_47 := ANY_TO_DINT(RESVAR_INT);
        _IO_QX0_1_48 := RESVAR_DINT;
        _IO_QX0_1_49 := ANY_TO_DINT(RESVAR_LINT);
        _IO_QX0_1_50 := ANY_TO_DINT(RESVAR_USINT);
        _IO_QX0_1_51 := ANY_TO_DINT(RESVAR_UINT);
        _IO_QX0_1_52 := RESVAR_UDINT;
        _IO_QX0_1_53 := ANY_TO_DINT(RESVAR_ULINT);
        _IO_QX0_1_54 := ANY_TO_DINT(RESVAR_REAL);
        _IO_QX0_1_55 := ANY_TO_DINT(RESVAR_LREAL);

        _IO_QX0_1_56 := ANY_TO_DINT(RESVAR_BYTE);
        _IO_QX0_1_57 := ANY_TO_DINT(RESVAR_WORD);
        _IO_QX0_1_58 := RESVAR_DWORD;
        _IO_QX0_1_59 := ANY_TO_DINT(RESVAR_LWORD);
        _IO_QX0_1_60 := ANY_TO_DINT(RESVAR_SINT);
        _IO_QX0_1_61 := ANY_TO_DINT(RESVAR_INT);
        _IO_QX0_1_62 := RESVAR_DINT;
        _IO_QX0_1_63 := ANY_TO_DINT(RESVAR_LINT);
        _IO_QX0_1_64 := ANY_TO_DINT(RESVAR_USINT);
        _IO_QX0_1_65 := ANY_TO_DINT(RESVAR_UINT);
        _IO_QX0_1_66 := RESVAR_UDINT;
        _IO_QX0_1_67 := ANY_TO_DINT(RESVAR_ULINT);
        _IO_QX0_1_68 := ANY_TO_DINT(RESVAR_REAL);
        _IO_QX0_1_69 := ANY_TO_DINT(RESVAR_LREAL);

        _IO_QX0_1_70 := ANY_TO_DINT(RESVAR_BYTE);
        _IO_QX0_1_71 := ANY_TO_DINT(RESVAR_WORD);
        _IO_QX0_1_72 := RESVAR_DWORD;
        _IO_QX0_1_73 := ANY_TO_DINT(RESVAR_LWORD);
        _IO_QX0_1_74 := ANY_TO_DINT(RESVAR_SINT);
        _IO_QX0_1_75 := ANY_TO_DINT(RESVAR_INT);
        _IO_QX0_1_76 := RESVAR_DINT;
        _IO_QX0_1_77 := ANY_TO_DINT(RESVAR_LINT);
        _IO_QX0_1_78 := ANY_TO_DINT(RESVAR_USINT);
        _IO_QX0_1_79 := ANY_TO_DINT(RESVAR_UINT);
        _IO_QX0_1_80 := RESVAR_UDINT;
        _IO_QX0_1_81 := ANY_TO_DINT(RESVAR_ULINT);
        _IO_QX0_1_82 := ANY_TO_DINT(RESVAR_REAL);
        _IO_QX0_1_83 := ANY_TO_DINT(RESVAR_LREAL);

        _IO_QX0_1_84 := ANY_TO_DINT(RESVAR_BYTE);
        _IO_QX0_1_85 := ANY_TO_DINT(RESVAR_WORD);
        _IO_QX0_1_86 := RESVAR_DWORD;
        _IO_QX0_1_87 := ANY_TO_DINT(RESVAR_LWORD);
        _IO_QX0_1_88 := ANY_TO_DINT(RESVAR_SINT);
        _IO_QX0_1_89 := ANY_TO_DINT(RESVAR_INT);
        _IO_QX0_1_90 := RESVAR_DINT;
        _IO_QX0_1_91 := ANY_TO_DINT(RESVAR_LINT);
        _IO_QX0_1_92 := ANY_TO_DINT(RESVAR_USINT);
        _IO_QX0_1_93 := ANY_TO_DINT(RESVAR_UINT);
        _IO_QX0_1_94 := RESVAR_UDINT;
        _IO_QX0_1_95 := ANY_TO_DINT(RESVAR_ULINT);
        _IO_QX0_1_96 := ANY_TO_DINT(RESVAR_REAL);
        _IO_QX0_1_97 := ANY_TO_DINT(RESVAR_LREAL);

    // Переменные REAL, регистры - 42000...51999
        _IO_QX8_1_0 := ANY_TO_REAL(RESVAR_BYTE);
        _IO_QX8_1_1 := ANY_TO_REAL(RESVAR_WORD);
        _IO_QX8_1_2 := ANY_TO_REAL(RESVAR_DWORD);
        _IO_QX8_1_3 := ANY_TO_REAL(RESVAR_LWORD);
        _IO_QX8_1_4 := ANY_TO_REAL(RESVAR_SINT);
        _IO_QX8_1_5 := ANY_TO_REAL(RESVAR_INT);
        _IO_QX8_1_6 := ANY_TO_REAL(RESVAR_DINT);
        _IO_QX8_1_7 := ANY_TO_REAL(RESVAR_LINT);
        _IO_QX8_1_8 := ANY_TO_REAL(RESVAR_USINT);
        _IO_QX8_1_9 := ANY_TO_REAL(RESVAR_UINT);
        _IO_QX8_1_10 := ANY_TO_REAL(RESVAR_UDINT);
        _IO_QX8_1_11 := ANY_TO_REAL(RESVAR_ULINT);
        _IO_QX8_1_12 := RESVAR_REAL;
        _IO_QX8_1_13 := ANY_TO_REAL(RESVAR_LREAL);

        _IO_QX8_1_14 := ANY_TO_REAL(RESVAR_BYTE);
        _IO_QX8_1_15 := ANY_TO_REAL(RESVAR_WORD);
        _IO_QX8_1_16 := ANY_TO_REAL(RESVAR_DWORD);
        _IO_QX8_1_17 := ANY_TO_REAL(RESVAR_LWORD);
        _IO_QX8_1_18 := ANY_TO_REAL(RESVAR_SINT);
        _IO_QX8_1_19 := ANY_TO_REAL(RESVAR_INT);
        _IO_QX8_1_20 := ANY_TO_REAL(RESVAR_DINT);
        _IO_QX8_1_21 := ANY_TO_REAL(RESVAR_LINT);
        _IO_QX8_1_22 := ANY_TO_REAL(RESVAR_USINT);
        _IO_QX8_1_23 := ANY_TO_REAL(RESVAR_UINT);
        _IO_QX8_1_24 := ANY_TO_REAL(RESVAR_UDINT);
        _IO_QX8_1_25 := ANY_TO_REAL(RESVAR_ULINT);
        _IO_QX8_1_26 := RESVAR_REAL;
        _IO_QX8_1_27 := ANY_TO_REAL(RESVAR_LREAL);

        _IO_QX8_1_28 := ANY_TO_REAL(RESVAR_BYTE);
        _IO_QX8_1_29 := ANY_TO_REAL(RESVAR_WORD);
        _IO_QX8_1_30 := ANY_TO_REAL(RESVAR_DWORD);
        _IO_QX8_1_31 := ANY_TO_REAL(RESVAR_LWORD);
        _IO_QX8_1_32 := ANY_TO_REAL(RESVAR_SINT);
        _IO_QX8_1_33 := ANY_TO_REAL(RESVAR_INT);
        _IO_QX8_1_34 := ANY_TO_REAL(RESVAR_DINT);
        _IO_QX8_1_35 := ANY_TO_REAL(RESVAR_LINT);
        _IO_QX8_1_36 := ANY_TO_REAL(RESVAR_USINT);
        _IO_QX8_1_37 := ANY_TO_REAL(RESVAR_UINT);
        _IO_QX8_1_38 := ANY_TO_REAL(RESVAR_UDINT);
        _IO_QX8_1_39 := ANY_TO_REAL(RESVAR_ULINT);
        _IO_QX8_1_40 := RESVAR_REAL;
        _IO_QX8_1_41 := ANY_TO_REAL(RESVAR_LREAL);

        _IO_QX8_1_42 := ANY_TO_REAL(RESVAR_BYTE);
        _IO_QX8_1_43 := ANY_TO_REAL(RESVAR_WORD);
        _IO_QX8_1_44 := ANY_TO_REAL(RESVAR_DWORD);
        _IO_QX8_1_45 := ANY_TO_REAL(RESVAR_LWORD);
        _IO_QX8_1_46 := ANY_TO_REAL(RESVAR_SINT);
        _IO_QX8_1_47 := ANY_TO_REAL(RESVAR_INT);
        _IO_QX8_1_48 := ANY_TO_REAL(RESVAR_DINT);
        _IO_QX8_1_49 := ANY_TO_REAL(RESVAR_LINT);
        _IO_QX8_1_50 := ANY_TO_REAL(RESVAR_USINT);
        _IO_QX8_1_51 := ANY_TO_REAL(RESVAR_UINT);
        _IO_QX8_1_52 := ANY_TO_REAL(RESVAR_UDINT);
        _IO_QX8_1_53 := ANY_TO_REAL(RESVAR_ULINT);
        _IO_QX8_1_54 := RESVAR_REAL;
        _IO_QX8_1_55 := ANY_TO_REAL(RESVAR_LREAL);

        _IO_QX8_1_56 := ANY_TO_REAL(RESVAR_BYTE);
        _IO_QX8_1_57 := ANY_TO_REAL(RESVAR_WORD);
        _IO_QX8_1_58 := ANY_TO_REAL(RESVAR_DWORD);
        _IO_QX8_1_59 := ANY_TO_REAL(RESVAR_LWORD);
        _IO_QX8_1_60 := ANY_TO_REAL(RESVAR_SINT);
        _IO_QX8_1_61 := ANY_TO_REAL(RESVAR_INT);
        _IO_QX8_1_62 := ANY_TO_REAL(RESVAR_DINT);
        _IO_QX8_1_63 := ANY_TO_REAL(RESVAR_LINT);
        _IO_QX8_1_64 := ANY_TO_REAL(RESVAR_USINT);
        _IO_QX8_1_65 := ANY_TO_REAL(RESVAR_UINT);
        _IO_QX8_1_66 := ANY_TO_REAL(RESVAR_UDINT);
        _IO_QX8_1_67 := ANY_TO_REAL(RESVAR_ULINT);
        _IO_QX8_1_68 := RESVAR_REAL;
        _IO_QX8_1_69 := ANY_TO_REAL(RESVAR_LREAL);

        _IO_QX8_1_70 := ANY_TO_REAL(RESVAR_BYTE);
        _IO_QX8_1_71 := ANY_TO_REAL(RESVAR_WORD);
        _IO_QX8_1_72 := ANY_TO_REAL(RESVAR_DWORD);
        _IO_QX8_1_73 := ANY_TO_REAL(RESVAR_LWORD);
        _IO_QX8_1_74 := ANY_TO_REAL(RESVAR_SINT);
        _IO_QX8_1_75 := ANY_TO_REAL(RESVAR_INT);
        _IO_QX8_1_76 := ANY_TO_REAL(RESVAR_DINT);
        _IO_QX8_1_77 := ANY_TO_REAL(RESVAR_LINT);
        _IO_QX8_1_78 := ANY_TO_REAL(RESVAR_USINT);
        _IO_QX8_1_79 := ANY_TO_REAL(RESVAR_UINT);
        _IO_QX8_1_80 := ANY_TO_REAL(RESVAR_UDINT);
        _IO_QX8_1_81 := ANY_TO_REAL(RESVAR_ULINT);
        _IO_QX8_1_82 := RESVAR_REAL;
        _IO_QX8_1_83 := ANY_TO_REAL(RESVAR_LREAL);

        _IO_QX8_1_84 := ANY_TO_REAL(RESVAR_BYTE);
        _IO_QX8_1_85 := ANY_TO_REAL(RESVAR_WORD);
        _IO_QX8_1_86 := ANY_TO_REAL(RESVAR_DWORD);
        _IO_QX8_1_87 := ANY_TO_REAL(RESVAR_LWORD);
        _IO_QX8_1_88 := ANY_TO_REAL(RESVAR_SINT);
        _IO_QX8_1_89 := ANY_TO_REAL(RESVAR_INT);
        _IO_QX8_1_90 := ANY_TO_REAL(RESVAR_DINT);
        _IO_QX8_1_91 := ANY_TO_REAL(RESVAR_LINT);
        _IO_QX8_1_92 := ANY_TO_REAL(RESVAR_USINT);
        _IO_QX8_1_93 := ANY_TO_REAL(RESVAR_UINT);
        _IO_QX8_1_94 := ANY_TO_REAL(RESVAR_UDINT);
        _IO_QX8_1_95 := ANY_TO_REAL(RESVAR_ULINT);
        _IO_QX8_1_96 := RESVAR_REAL;
        _IO_QX8_1_97 := ANY_TO_REAL(RESVAR_LREAL);

    // Переменные INT, регистры - 52000...61999
        _IO_QX9_1_0 := ANY_TO_DINT(RESVAR_BYTE);
        _IO_QX9_1_1 := ANY_TO_DINT(RESVAR_WORD);
        _IO_QX9_1_2 := RESVAR_DWORD;
        _IO_QX9_1_3 := ANY_TO_DINT(RESVAR_LWORD);
        _IO_QX9_1_4 := ANY_TO_DINT(RESVAR_SINT);
        _IO_QX9_1_5 := ANY_TO_DINT(RESVAR_INT);
        _IO_QX9_1_6 := RESVAR_DINT;
        _IO_QX9_1_7 := ANY_TO_DINT(RESVAR_LINT);
        _IO_QX9_1_8 := ANY_TO_DINT(RESVAR_USINT);
        _IO_QX9_1_9 := ANY_TO_DINT(RESVAR_UINT);
        _IO_QX9_1_10 := RESVAR_UDINT;
        _IO_QX9_1_11 := ANY_TO_DINT(RESVAR_ULINT);
        _IO_QX9_1_12 := ANY_TO_DINT(RESVAR_REAL);
        _IO_QX9_1_13 := ANY_TO_DINT(RESVAR_LREAL);

        _IO_QX9_1_14 := ANY_TO_DINT(RESVAR_BYTE);
        _IO_QX9_1_15 := ANY_TO_DINT(RESVAR_WORD);
        _IO_QX9_1_16 := RESVAR_DWORD;
        _IO_QX9_1_17 := ANY_TO_DINT(RESVAR_LWORD);
        _IO_QX9_1_18 := ANY_TO_DINT(RESVAR_SINT);
        _IO_QX9_1_19 := ANY_TO_DINT(RESVAR_INT);
        _IO_QX9_1_20 := RESVAR_DINT;
        _IO_QX9_1_21 := ANY_TO_DINT(RESVAR_LINT);
        _IO_QX9_1_22 := ANY_TO_DINT(RESVAR_USINT);
        _IO_QX9_1_23 := ANY_TO_DINT(RESVAR_UINT);
        _IO_QX9_1_24 := RESVAR_UDINT;
        _IO_QX9_1_25 := ANY_TO_DINT(RESVAR_ULINT);
        _IO_QX9_1_26 := ANY_TO_DINT(RESVAR_REAL);
        _IO_QX9_1_27 := ANY_TO_DINT(RESVAR_LREAL);

        _IO_QX9_1_28 := ANY_TO_DINT(RESVAR_BYTE);
        _IO_QX9_1_29 := ANY_TO_DINT(RESVAR_WORD);
        _IO_QX9_1_30 := RESVAR_DWORD;
        _IO_QX9_1_31 := ANY_TO_DINT(RESVAR_LWORD);
        _IO_QX9_1_32 := ANY_TO_DINT(RESVAR_SINT);
        _IO_QX9_1_33 := ANY_TO_DINT(RESVAR_INT);
        _IO_QX9_1_34 := RESVAR_DINT;
        _IO_QX9_1_35 := ANY_TO_DINT(RESVAR_LINT);
        _IO_QX9_1_36 := ANY_TO_DINT(RESVAR_USINT);
        _IO_QX9_1_37 := ANY_TO_DINT(RESVAR_UINT);
        _IO_QX9_1_38 := RESVAR_UDINT;
        _IO_QX9_1_39 := ANY_TO_DINT(RESVAR_ULINT);
        _IO_QX9_1_40 := ANY_TO_DINT(RESVAR_REAL);
        _IO_QX9_1_41 := ANY_TO_DINT(RESVAR_LREAL);

        _IO_QX9_1_42 := ANY_TO_DINT(RESVAR_BYTE);
        _IO_QX9_1_43 := ANY_TO_DINT(RESVAR_WORD);
        _IO_QX9_1_44 := RESVAR_DWORD;
        _IO_QX9_1_45 := ANY_TO_DINT(RESVAR_LWORD);
        _IO_QX9_1_46 := ANY_TO_DINT(RESVAR_SINT);
        _IO_QX9_1_47 := ANY_TO_DINT(RESVAR_INT);
        _IO_QX9_1_48 := RESVAR_DINT;
        _IO_QX9_1_49 := ANY_TO_DINT(RESVAR_LINT);
        _IO_QX9_1_50 := ANY_TO_DINT(RESVAR_USINT);
        _IO_QX9_1_51 := ANY_TO_DINT(RESVAR_UINT);
        _IO_QX9_1_52 := RESVAR_UDINT;
        _IO_QX9_1_53 := ANY_TO_DINT(RESVAR_ULINT);
        _IO_QX9_1_54 := ANY_TO_DINT(RESVAR_REAL);
        _IO_QX9_1_55 := ANY_TO_DINT(RESVAR_LREAL);

        _IO_QX9_1_56 := ANY_TO_DINT(RESVAR_BYTE);
        _IO_QX9_1_57 := ANY_TO_DINT(RESVAR_WORD);
        _IO_QX9_1_58 := RESVAR_DWORD;
        _IO_QX9_1_59 := ANY_TO_DINT(RESVAR_LWORD);
        _IO_QX9_1_60 := ANY_TO_DINT(RESVAR_SINT);
        _IO_QX9_1_61 := ANY_TO_DINT(RESVAR_INT);
        _IO_QX9_1_62 := RESVAR_DINT;
        _IO_QX9_1_63 := ANY_TO_DINT(RESVAR_LINT);
        _IO_QX9_1_64 := ANY_TO_DINT(RESVAR_USINT);
        _IO_QX9_1_65 := ANY_TO_DINT(RESVAR_UINT);
        _IO_QX9_1_66 := RESVAR_UDINT;
        _IO_QX9_1_67 := ANY_TO_DINT(RESVAR_ULINT);
        _IO_QX9_1_68 := ANY_TO_DINT(RESVAR_REAL);
        _IO_QX9_1_69 := ANY_TO_DINT(RESVAR_LREAL);

        _IO_QX9_1_70 := ANY_TO_DINT(RESVAR_BYTE);
        _IO_QX9_1_71 := ANY_TO_DINT(RESVAR_WORD);
        _IO_QX9_1_72 := RESVAR_DWORD;
        _IO_QX9_1_73 := ANY_TO_DINT(RESVAR_LWORD);
        _IO_QX9_1_74 := ANY_TO_DINT(RESVAR_SINT);
        _IO_QX9_1_75 := ANY_TO_DINT(RESVAR_INT);
        _IO_QX9_1_76 := RESVAR_DINT;
        _IO_QX9_1_77 := ANY_TO_DINT(RESVAR_LINT);
        _IO_QX9_1_78 := ANY_TO_DINT(RESVAR_USINT);
        _IO_QX9_1_79 := ANY_TO_DINT(RESVAR_UINT);
        _IO_QX9_1_80 := RESVAR_UDINT;
        _IO_QX9_1_81 := ANY_TO_DINT(RESVAR_ULINT);
        _IO_QX9_1_82 := ANY_TO_DINT(RESVAR_REAL);
        _IO_QX9_1_83 := ANY_TO_DINT(RESVAR_LREAL);

        _IO_QX9_1_84 := ANY_TO_DINT(RESVAR_BYTE);
        _IO_QX9_1_85 := ANY_TO_DINT(RESVAR_WORD);
        _IO_QX9_1_86 := RESVAR_DWORD;
        _IO_QX9_1_87 := ANY_TO_DINT(RESVAR_LWORD);
        _IO_QX9_1_88 := ANY_TO_DINT(RESVAR_SINT);
        _IO_QX9_1_89 := ANY_TO_DINT(RESVAR_INT);
        _IO_QX9_1_90 := RESVAR_DINT;
        _IO_QX9_1_91 := ANY_TO_DINT(RESVAR_LINT);
        _IO_QX9_1_92 := ANY_TO_DINT(RESVAR_USINT);
        _IO_QX9_1_93 := ANY_TO_DINT(RESVAR_UINT);
        _IO_QX9_1_94 := RESVAR_UDINT;
        _IO_QX9_1_95 := ANY_TO_DINT(RESVAR_ULINT);
        _IO_QX9_1_96 := ANY_TO_DINT(RESVAR_REAL);
        _IO_QX9_1_97 := ANY_TO_DINT(RESVAR_LREAL);

(* Считывание IR регистров *)
    // Переменные DINT, регистры - 32000...41999
        _IO_QU2_0 := ANY_TO_DINT(RESVAR_BYTE);
        _IO_QU2_1 := ANY_TO_DINT(RESVAR_WORD);
        _IO_QU2_2 := RESVAR_DWORD;
        _IO_QU2_3 := ANY_TO_DINT(RESVAR_LWORD);
        _IO_QU2_4 := ANY_TO_DINT(RESVAR_SINT);
        _IO_QU2_5 := ANY_TO_DINT(RESVAR_INT);
        _IO_QU2_6 := RESVAR_DINT;
        _IO_QU2_7 := ANY_TO_DINT(RESVAR_LINT);
        _IO_QU2_8 := ANY_TO_DINT(RESVAR_USINT);
        _IO_QU2_9 := ANY_TO_DINT(RESVAR_UINT);
        _IO_QU2_10 := RESVAR_UDINT;
        _IO_QU2_11 := ANY_TO_DINT(RESVAR_ULINT);
        _IO_QU2_12 := ANY_TO_DINT(RESVAR_REAL);
        _IO_QU2_13 := ANY_TO_DINT(RESVAR_LREAL);

        _IO_QU2_14 := ANY_TO_DINT(RESVAR_BYTE);
        _IO_QU2_15 := ANY_TO_DINT(RESVAR_WORD);
        _IO_QU2_16 := RESVAR_DWORD;
        _IO_QU2_17 := ANY_TO_DINT(RESVAR_LWORD);
        _IO_QU2_18 := ANY_TO_DINT(RESVAR_SINT);
        _IO_QU2_19 := ANY_TO_DINT(RESVAR_INT);
        _IO_QU2_20 := RESVAR_DINT;
        _IO_QU2_21 := ANY_TO_DINT(RESVAR_LINT);
        _IO_QU2_22 := ANY_TO_DINT(RESVAR_USINT);
        _IO_QU2_23 := ANY_TO_DINT(RESVAR_UINT);
        _IO_QU2_24 := RESVAR_UDINT;
        _IO_QU2_25 := ANY_TO_DINT(RESVAR_ULINT);
        _IO_QU2_26 := ANY_TO_DINT(RESVAR_REAL);
        _IO_QU2_27 := ANY_TO_DINT(RESVAR_LREAL);

        _IO_QU2_28 := ANY_TO_DINT(RESVAR_BYTE);
        _IO_QU2_29 := ANY_TO_DINT(RESVAR_WORD);
        _IO_QU2_30 := RESVAR_DWORD;
        _IO_QU2_31 := ANY_TO_DINT(RESVAR_LWORD);
        _IO_QU2_32 := ANY_TO_DINT(RESVAR_SINT);
        _IO_QU2_33 := ANY_TO_DINT(RESVAR_INT);
        _IO_QU2_34 := RESVAR_DINT;
        _IO_QU2_35 := ANY_TO_DINT(RESVAR_LINT);
        _IO_QU2_36 := ANY_TO_DINT(RESVAR_USINT);
        _IO_QU2_37 := ANY_TO_DINT(RESVAR_UINT);
        _IO_QU2_38 := RESVAR_UDINT;
        _IO_QU2_39 := ANY_TO_DINT(RESVAR_ULINT);
        _IO_QU2_40 := ANY_TO_DINT(RESVAR_REAL);
        _IO_QU2_41 := ANY_TO_DINT(RESVAR_LREAL);

        _IO_QU2_42 := ANY_TO_DINT(RESVAR_BYTE);
        _IO_QU2_43 := ANY_TO_DINT(RESVAR_WORD);
        _IO_QU2_44 := RESVAR_DWORD;
        _IO_QU2_45 := ANY_TO_DINT(RESVAR_LWORD);
        _IO_QU2_46 := ANY_TO_DINT(RESVAR_SINT);
        _IO_QU2_47 := ANY_TO_DINT(RESVAR_INT);
        _IO_QU2_48 := RESVAR_DINT;
        _IO_QU2_49 := ANY_TO_DINT(RESVAR_LINT);
        _IO_QU2_50 := ANY_TO_DINT(RESVAR_USINT);
        _IO_QU2_51 := ANY_TO_DINT(RESVAR_UINT);
        _IO_QU2_52 := RESVAR_UDINT;
        _IO_QU2_53 := ANY_TO_DINT(RESVAR_ULINT);
        _IO_QU2_54 := ANY_TO_DINT(RESVAR_REAL);
        _IO_QU2_55 := ANY_TO_DINT(RESVAR_LREAL);

        _IO_QU2_56 := ANY_TO_DINT(RESVAR_BYTE);
        _IO_QU2_57 := ANY_TO_DINT(RESVAR_WORD);
        _IO_QU2_58 := RESVAR_DWORD;
        _IO_QU2_59 := ANY_TO_DINT(RESVAR_LWORD);
        _IO_QU2_60 := ANY_TO_DINT(RESVAR_SINT);
        _IO_QU2_61 := ANY_TO_DINT(RESVAR_INT);
        _IO_QU2_62 := RESVAR_DINT;
        _IO_QU2_63 := ANY_TO_DINT(RESVAR_LINT);
        _IO_QU2_64 := ANY_TO_DINT(RESVAR_USINT);
        _IO_QU2_65 := ANY_TO_DINT(RESVAR_UINT);
        _IO_QU2_66 := RESVAR_UDINT;
        _IO_QU2_67 := ANY_TO_DINT(RESVAR_ULINT);
        _IO_QU2_68 := ANY_TO_DINT(RESVAR_REAL);
        _IO_QU2_69 := ANY_TO_DINT(RESVAR_LREAL);

        _IO_QU2_70 := ANY_TO_DINT(RESVAR_BYTE);
        _IO_QU2_71 := ANY_TO_DINT(RESVAR_WORD);
        _IO_QU2_72 := RESVAR_DWORD;
        _IO_QU2_73 := ANY_TO_DINT(RESVAR_LWORD);
        _IO_QU2_74 := ANY_TO_DINT(RESVAR_SINT);
        _IO_QU2_75 := ANY_TO_DINT(RESVAR_INT);
        _IO_QU2_76 := RESVAR_DINT;
        _IO_QU2_77 := ANY_TO_DINT(RESVAR_LINT);
        _IO_QU2_78 := ANY_TO_DINT(RESVAR_USINT);
        _IO_QU2_79 := ANY_TO_DINT(RESVAR_UINT);
        _IO_QU2_80 := RESVAR_UDINT;
        _IO_QU2_81 := ANY_TO_DINT(RESVAR_ULINT);
        _IO_QU2_82 := ANY_TO_DINT(RESVAR_REAL);
        _IO_QU2_83 := ANY_TO_DINT(RESVAR_LREAL);

        _IO_QU2_84 := ANY_TO_DINT(RESVAR_BYTE);
        _IO_QU2_85 := ANY_TO_DINT(RESVAR_WORD);
        _IO_QU2_86 := RESVAR_DWORD;
        _IO_QU2_87 := ANY_TO_DINT(RESVAR_LWORD);
        _IO_QU2_88 := ANY_TO_DINT(RESVAR_SINT);
        _IO_QU2_89 := ANY_TO_DINT(RESVAR_INT);
        _IO_QU2_90 := RESVAR_DINT;
        _IO_QU2_91 := ANY_TO_DINT(RESVAR_LINT);
        _IO_QU2_92 := ANY_TO_DINT(RESVAR_USINT);
        _IO_QU2_93 := ANY_TO_DINT(RESVAR_UINT);
        _IO_QU2_94 := RESVAR_UDINT;
        _IO_QU2_95 := ANY_TO_DINT(RESVAR_ULINT);
        _IO_QU2_96 := ANY_TO_DINT(RESVAR_REAL);
        _IO_QU2_97 := ANY_TO_DINT(RESVAR_LREAL);

    // Переменные REAL, регистры - 42000...51999
        _IO_QU3_0 := ANY_TO_REAL(RESVAR_BYTE);
        _IO_QU3_1 := ANY_TO_REAL(RESVAR_WORD);
        _IO_QU3_2 := ANY_TO_REAL(RESVAR_DWORD);
        _IO_QU3_3 := ANY_TO_REAL(RESVAR_LWORD);
        _IO_QU3_4 := ANY_TO_REAL(RESVAR_SINT);
        _IO_QU3_5 := ANY_TO_REAL(RESVAR_INT);
        _IO_QU3_6 := ANY_TO_REAL(RESVAR_DINT);
        _IO_QU3_7 := ANY_TO_REAL(RESVAR_LINT);
        _IO_QU3_8 := ANY_TO_REAL(RESVAR_USINT);
        _IO_QU3_9 := ANY_TO_REAL(RESVAR_UINT);
        _IO_QU3_10 := ANY_TO_REAL(RESVAR_UDINT);
        _IO_QU3_11 := ANY_TO_REAL(RESVAR_ULINT);
        _IO_QU3_12 := RESVAR_REAL;
        _IO_QU3_13 := ANY_TO_REAL(RESVAR_LREAL);

        _IO_QU3_14 := ANY_TO_REAL(RESVAR_BYTE);
        _IO_QU3_15 := ANY_TO_REAL(RESVAR_WORD);
        _IO_QU3_16 := ANY_TO_REAL(RESVAR_DWORD);
        _IO_QU3_17 := ANY_TO_REAL(RESVAR_LWORD);
        _IO_QU3_18 := ANY_TO_REAL(RESVAR_SINT);
        _IO_QU3_19 := ANY_TO_REAL(RESVAR_INT);
        _IO_QU3_20 := ANY_TO_REAL(RESVAR_DINT);
        _IO_QU3_21 := ANY_TO_REAL(RESVAR_LINT);
        _IO_QU3_22 := ANY_TO_REAL(RESVAR_USINT);
        _IO_QU3_23 := ANY_TO_REAL(RESVAR_UINT);
        _IO_QU3_24 := ANY_TO_REAL(RESVAR_UDINT);
        _IO_QU3_25 := ANY_TO_REAL(RESVAR_ULINT);
        _IO_QU3_26 := RESVAR_REAL;
        _IO_QU3_27 := ANY_TO_REAL(RESVAR_LREAL);

        _IO_QU3_28 := ANY_TO_REAL(RESVAR_BYTE);
        _IO_QU3_29 := ANY_TO_REAL(RESVAR_WORD);
        _IO_QU3_30 := ANY_TO_REAL(RESVAR_DWORD);
        _IO_QU3_31 := ANY_TO_REAL(RESVAR_LWORD);
        _IO_QU3_32 := ANY_TO_REAL(RESVAR_SINT);
        _IO_QU3_33 := ANY_TO_REAL(RESVAR_INT);
        _IO_QU3_34 := ANY_TO_REAL(RESVAR_DINT);
        _IO_QU3_35 := ANY_TO_REAL(RESVAR_LINT);
        _IO_QU3_36 := ANY_TO_REAL(RESVAR_USINT);
        _IO_QU3_37 := ANY_TO_REAL(RESVAR_UINT);
        _IO_QU3_38 := ANY_TO_REAL(RESVAR_UDINT);
        _IO_QU3_39 := ANY_TO_REAL(RESVAR_ULINT);
        _IO_QU3_40 := RESVAR_REAL;
        _IO_QU3_41 := ANY_TO_REAL(RESVAR_LREAL);

        _IO_QU3_42 := ANY_TO_REAL(RESVAR_BYTE);
        _IO_QU3_43 := ANY_TO_REAL(RESVAR_WORD);
        _IO_QU3_44 := ANY_TO_REAL(RESVAR_DWORD);
        _IO_QU3_45 := ANY_TO_REAL(RESVAR_LWORD);
        _IO_QU3_46 := ANY_TO_REAL(RESVAR_SINT);
        _IO_QU3_47 := ANY_TO_REAL(RESVAR_INT);
        _IO_QU3_48 := ANY_TO_REAL(RESVAR_DINT);
        _IO_QU3_49 := ANY_TO_REAL(RESVAR_LINT);
        _IO_QU3_50 := ANY_TO_REAL(RESVAR_USINT);
        _IO_QU3_51 := ANY_TO_REAL(RESVAR_UINT);
        _IO_QU3_52 := ANY_TO_REAL(RESVAR_UDINT);
        _IO_QU3_53 := ANY_TO_REAL(RESVAR_ULINT);
        _IO_QU3_54 := RESVAR_REAL;
        _IO_QU3_55 := ANY_TO_REAL(RESVAR_LREAL);

        _IO_QU3_56 := ANY_TO_REAL(RESVAR_BYTE);
        _IO_QU3_57 := ANY_TO_REAL(RESVAR_WORD);
        _IO_QU3_58 := ANY_TO_REAL(RESVAR_DWORD);
        _IO_QU3_59 := ANY_TO_REAL(RESVAR_LWORD);
        _IO_QU3_60 := ANY_TO_REAL(RESVAR_SINT);
        _IO_QU3_61 := ANY_TO_REAL(RESVAR_INT);
        _IO_QU3_62 := ANY_TO_REAL(RESVAR_DINT);
        _IO_QU3_63 := ANY_TO_REAL(RESVAR_LINT);
        _IO_QU3_64 := ANY_TO_REAL(RESVAR_USINT);
        _IO_QU3_65 := ANY_TO_REAL(RESVAR_UINT);
        _IO_QU3_66 := ANY_TO_REAL(RESVAR_UDINT);
        _IO_QU3_67 := ANY_TO_REAL(RESVAR_ULINT);
        _IO_QU3_68 := RESVAR_REAL;
        _IO_QU3_69 := ANY_TO_REAL(RESVAR_LREAL);

        _IO_QU3_70 := ANY_TO_REAL(RESVAR_BYTE);
        _IO_QU3_71 := ANY_TO_REAL(RESVAR_WORD);
        _IO_QU3_72 := ANY_TO_REAL(RESVAR_DWORD);
        _IO_QU3_73 := ANY_TO_REAL(RESVAR_LWORD);
        _IO_QU3_74 := ANY_TO_REAL(RESVAR_SINT);
        _IO_QU3_75 := ANY_TO_REAL(RESVAR_INT);
        _IO_QU3_76 := ANY_TO_REAL(RESVAR_DINT);
        _IO_QU3_77 := ANY_TO_REAL(RESVAR_LINT);
        _IO_QU3_78 := ANY_TO_REAL(RESVAR_USINT);
        _IO_QU3_79 := ANY_TO_REAL(RESVAR_UINT);
        _IO_QU3_80 := ANY_TO_REAL(RESVAR_UDINT);
        _IO_QU3_81 := ANY_TO_REAL(RESVAR_ULINT);
        _IO_QU3_82 := RESVAR_REAL;
        _IO_QU3_83 := ANY_TO_REAL(RESVAR_LREAL);

        _IO_QU3_84 := ANY_TO_REAL(RESVAR_BYTE);
        _IO_QU3_85 := ANY_TO_REAL(RESVAR_WORD);
        _IO_QU3_86 := ANY_TO_REAL(RESVAR_DWORD);
        _IO_QU3_87 := ANY_TO_REAL(RESVAR_LWORD);
        _IO_QU3_88 := ANY_TO_REAL(RESVAR_SINT);
        _IO_QU3_89 := ANY_TO_REAL(RESVAR_INT);
        _IO_QU3_90 := ANY_TO_REAL(RESVAR_DINT);
        _IO_QU3_91 := ANY_TO_REAL(RESVAR_LINT);
        _IO_QU3_92 := ANY_TO_REAL(RESVAR_USINT);
        _IO_QU3_93 := ANY_TO_REAL(RESVAR_UINT);
        _IO_QU3_94 := ANY_TO_REAL(RESVAR_UDINT);
        _IO_QU3_95 := ANY_TO_REAL(RESVAR_ULINT);
        _IO_QU3_96 := RESVAR_REAL;
        _IO_QU3_97 := ANY_TO_REAL(RESVAR_LREAL);

    // Переменные INT, регистры - 52000...61999
        _IO_QU4_0 := ANY_TO_DINT(RESVAR_BYTE);
        _IO_QU4_1 := ANY_TO_DINT(RESVAR_WORD);
        _IO_QU4_2 := RESVAR_DWORD;
        _IO_QU4_3 := ANY_TO_DINT(RESVAR_LWORD);
        _IO_QU4_4 := ANY_TO_DINT(RESVAR_SINT);
        _IO_QU4_5 := ANY_TO_DINT(RESVAR_INT);
        _IO_QU4_6 := RESVAR_DINT;
        _IO_QU4_7 := ANY_TO_DINT(RESVAR_LINT);
        _IO_QU4_8 := ANY_TO_DINT(RESVAR_USINT);
        _IO_QU4_9 := ANY_TO_DINT(RESVAR_UINT);
        _IO_QU4_10 := RESVAR_UDINT;
        _IO_QU4_11 := ANY_TO_DINT(RESVAR_ULINT);
        _IO_QU4_12 := ANY_TO_DINT(RESVAR_REAL);
        _IO_QU4_13 := ANY_TO_DINT(RESVAR_LREAL);

        _IO_QU4_14 := ANY_TO_DINT(RESVAR_BYTE);
        _IO_QU4_15 := ANY_TO_DINT(RESVAR_WORD);
        _IO_QU4_16 := RESVAR_DWORD;
        _IO_QU4_17 := ANY_TO_DINT(RESVAR_LWORD);
        _IO_QU4_18 := ANY_TO_DINT(RESVAR_SINT);
        _IO_QU4_19 := ANY_TO_DINT(RESVAR_INT);
        _IO_QU4_20 := RESVAR_DINT;
        _IO_QU4_21 := ANY_TO_DINT(RESVAR_LINT);
        _IO_QU4_22 := ANY_TO_DINT(RESVAR_USINT);
        _IO_QU4_23 := ANY_TO_DINT(RESVAR_UINT);
        _IO_QU4_24 := RESVAR_UDINT;
        _IO_QU4_25 := ANY_TO_DINT(RESVAR_ULINT);
        _IO_QU4_26 := ANY_TO_DINT(RESVAR_REAL);
        _IO_QU4_27 := ANY_TO_DINT(RESVAR_LREAL);

        _IO_QU4_28 := ANY_TO_DINT(RESVAR_BYTE);
        _IO_QU4_29 := ANY_TO_DINT(RESVAR_WORD);
        _IO_QU4_30 := RESVAR_DWORD;
        _IO_QU4_31 := ANY_TO_DINT(RESVAR_LWORD);
        _IO_QU4_32 := ANY_TO_DINT(RESVAR_SINT);
        _IO_QU4_33 := ANY_TO_DINT(RESVAR_INT);
        _IO_QU4_34 := RESVAR_DINT;
        _IO_QU4_35 := ANY_TO_DINT(RESVAR_LINT);
        _IO_QU4_36 := ANY_TO_DINT(RESVAR_USINT);
        _IO_QU4_37 := ANY_TO_DINT(RESVAR_UINT);
        _IO_QU4_38 := RESVAR_UDINT;
        _IO_QU4_39 := ANY_TO_DINT(RESVAR_ULINT);
        _IO_QU4_40 := ANY_TO_DINT(RESVAR_REAL);
        _IO_QU4_41 := ANY_TO_DINT(RESVAR_LREAL);

        _IO_QU4_42 := ANY_TO_DINT(RESVAR_BYTE);
        _IO_QU4_43 := ANY_TO_DINT(RESVAR_WORD);
        _IO_QU4_44 := RESVAR_DWORD;
        _IO_QU4_45 := ANY_TO_DINT(RESVAR_LWORD);
        _IO_QU4_46 := ANY_TO_DINT(RESVAR_SINT);
        _IO_QU4_47 := ANY_TO_DINT(RESVAR_INT);
        _IO_QU4_48 := RESVAR_DINT;
        _IO_QU4_49 := ANY_TO_DINT(RESVAR_LINT);
        _IO_QU4_50 := ANY_TO_DINT(RESVAR_USINT);
        _IO_QU4_51 := ANY_TO_DINT(RESVAR_UINT);
        _IO_QU4_52 := RESVAR_UDINT;
        _IO_QU4_53 := ANY_TO_DINT(RESVAR_ULINT);
        _IO_QU4_54 := ANY_TO_DINT(RESVAR_REAL);
        _IO_QU4_55 := ANY_TO_DINT(RESVAR_LREAL);

        _IO_QU4_56 := ANY_TO_DINT(RESVAR_BYTE);
        _IO_QU4_57 := ANY_TO_DINT(RESVAR_WORD);
        _IO_QU4_58 := RESVAR_DWORD;
        _IO_QU4_59 := ANY_TO_DINT(RESVAR_LWORD);
        _IO_QU4_60 := ANY_TO_DINT(RESVAR_SINT);
        _IO_QU4_61 := ANY_TO_DINT(RESVAR_INT);
        _IO_QU4_62 := RESVAR_DINT;
        _IO_QU4_63 := ANY_TO_DINT(RESVAR_LINT);
        _IO_QU4_64 := ANY_TO_DINT(RESVAR_USINT);
        _IO_QU4_65 := ANY_TO_DINT(RESVAR_UINT);
        _IO_QU4_66 := RESVAR_UDINT;
        _IO_QU4_67 := ANY_TO_DINT(RESVAR_ULINT);
        _IO_QU4_68 := ANY_TO_DINT(RESVAR_REAL);
        _IO_QU4_69 := ANY_TO_DINT(RESVAR_LREAL);

        _IO_QU4_70 := ANY_TO_DINT(RESVAR_BYTE);
        _IO_QU4_71 := ANY_TO_DINT(RESVAR_WORD);
        _IO_QU4_72 := RESVAR_DWORD;
        _IO_QU4_73 := ANY_TO_DINT(RESVAR_LWORD);
        _IO_QU4_74 := ANY_TO_DINT(RESVAR_SINT);
        _IO_QU4_75 := ANY_TO_DINT(RESVAR_INT);
        _IO_QU4_76 := RESVAR_DINT;
        _IO_QU4_77 := ANY_TO_DINT(RESVAR_LINT);
        _IO_QU4_78 := ANY_TO_DINT(RESVAR_USINT);
        _IO_QU4_79 := ANY_TO_DINT(RESVAR_UINT);
        _IO_QU4_80 := RESVAR_UDINT;
        _IO_QU4_81 := ANY_TO_DINT(RESVAR_ULINT);
        _IO_QU4_82 := ANY_TO_DINT(RESVAR_REAL);
        _IO_QU4_83 := ANY_TO_DINT(RESVAR_LREAL);

        _IO_QU4_84 := ANY_TO_DINT(RESVAR_BYTE);
        _IO_QU4_85 := ANY_TO_DINT(RESVAR_WORD);
        _IO_QU4_86 := RESVAR_DWORD;
        _IO_QU4_87 := ANY_TO_DINT(RESVAR_LWORD);
        _IO_QU4_88 := ANY_TO_DINT(RESVAR_SINT);
        _IO_QU4_89 := ANY_TO_DINT(RESVAR_INT);
        _IO_QU4_90 := RESVAR_DINT;
        _IO_QU4_91 := ANY_TO_DINT(RESVAR_LINT);
        _IO_QU4_92 := ANY_TO_DINT(RESVAR_USINT);
        _IO_QU4_93 := ANY_TO_DINT(RESVAR_UINT);
        _IO_QU4_94 := RESVAR_UDINT;
        _IO_QU4_95 := ANY_TO_DINT(RESVAR_ULINT);
        _IO_QU4_96 := ANY_TO_DINT(RESVAR_REAL);
        _IO_QU4_97 := ANY_TO_DINT(RESVAR_LREAL);

END_PROGRAM

(* ---- PRG HART_PULL_v1.st ---- *)
PROGRAM HART_PULL_v1

(* Программа опроса устройств по HART-протоколу *)

(* В программе происходит поочерёдное переключение команд запроса/чтения *)
(* Команда опроса переключается по временному интервалу *)
(* Ошибки опроса не учитываются при переключении команды опроса *)

// Конфигурация FB HART_Communication
HART_BUS := 1;
HART_DEVICE := 2;
HART_CHANNEL := 3;
HART_TIMEOUT := 500;

// Настройка таймера реального времени
// TIME_RV - экземпляр FB IMPRV
TIME_RV.W := FALSE;                                              // Режим работы: FALSE - периодический, TRUE - одиночный
TIME_RV.Nh := 0;
TIME_RV.Nm := 0;
TIME_RV.Ns := TIME_PULL;
TIME_RV.Timp := _PRESET_CYCLE_TIME;
TIME_RV ();

// Инициализация опроса
IF REQUEST AND TIME_RV.Out THEN

    // Приращение номера ветвления
    STEP_PULL := STEP_PULL + 1;

    CASE STEP_PULL OF

        1:  (* Функция 0 - чтение уникального идентификатора/адреса устройства *)
            FINAL_PULL := FALSE;
            HART_COMM_54.Request := FALSE;

            HART_COMM_00.Request := TRUE;
            HART_COMM_00.Bus := HART_BUS;
            HART_COMM_00.Device := HART_DEVICE;
            HART_COMM_00.Channel := HART_CHANNEL;
            HART_COMM_00.TimeOut := HART_TIMEOUT;

            // HART_FUNC := 'Функция 0';
            HART_FUNCTIONS := 0;

        2:  (* Функция 1 - чтение первичной переменной *)
            HART_COMM_00.Request := FALSE;

            HART_COMM_01.Request := TRUE;
            HART_COMM_01.Bus := HART_BUS;
            HART_COMM_01.Device := HART_DEVICE;
            HART_COMM_01.Channel := HART_CHANNEL;
            HART_COMM_01.TimeOut := HART_TIMEOUT;

            // HART_FUNC := 'Функция 1';
            HART_FUNCTIONS := 1;

        3:  (* Функция 2 - чтение первичной переменной как величины тока и в процентах от диапазона *)
            HART_COMM_01.Request := FALSE;

            HART_COMM_02.Request := TRUE;
            HART_COMM_02.Bus := HART_BUS;
            HART_COMM_02.Device := HART_DEVICE;
            HART_COMM_02.Channel := HART_CHANNEL;
            HART_COMM_02.TimeOut := HART_TIMEOUT;

            HART_FUNC := 'Функция 2';
            HART_FUNCTIONS := 2;

        4:  (* Функция 3 - чтение динамических переменных и токового значения первичной переменной *)
            HART_COMM_02.Request := FALSE;

            HART_COMM_03.Request := TRUE;
            HART_COMM_03.Bus := HART_BUS;
            HART_COMM_03.Device := HART_DEVICE;
            HART_COMM_03.Channel := HART_CHANNEL;
            HART_COMM_03.TimeOut := HART_TIMEOUT;

            // HART_FUNC := 'Функция 3';
            HART_FUNCTIONS := 3;

        5:  (* Функция 6 - запись адреса устройства *)
            HART_COMM_03.Request := FALSE;
            HART_COMM_06.Request := TRUE;

            HART_COMM_06.Request := TRUE;
            HART_COMM_06.Bus := HART_BUS;
            HART_COMM_06.Device := HART_DEVICE;
            HART_COMM_06.Channel := HART_CHANNEL;
            HART_COMM_06.TimeOut := HART_TIMEOUT;

            HART_FUNC := 'Функция 6';
            HART_FUNCTIONS := 6;

        6:  (* Функция 12 - чтение сообщения, содержащегося в устройстве *)
            HART_COMM_06.Request := FALSE;

            HART_COMM_12.Request := TRUE;
            HART_COMM_12.Bus := HART_BUS;
            HART_COMM_12.Device := HART_DEVICE;
            HART_COMM_12.Channel := HART_CHANNEL;
            HART_COMM_12.TimeOut := HART_TIMEOUT;

            // HART_FUNC := 'Функция 12';
            HART_FUNCTIONS := 12;

        7:  (* Функция 13 - чтение текстового тега, описателя и даты *)
            HART_COMM_12.Request := FALSE;

            HART_COMM_13.Request := TRUE;
            HART_COMM_13.Bus := HART_BUS;
            HART_COMM_13.Device := HART_DEVICE;
            HART_COMM_13.Channel := HART_CHANNEL;
            HART_COMM_13.TimeOut := HART_TIMEOUT;

            // HART_FUNC := 'Функция 13';
            HART_FUNCTIONS := 13;

        8:  (* Функция 14 - чтение информации сенсора первичной переменной *)
            HART_COMM_13.Request := FALSE;

            HART_COMM_14.Request := TRUE;
            HART_COMM_14.Bus := HART_BUS;
            HART_COMM_14.Device := HART_DEVICE;
            HART_COMM_14.Channel := HART_CHANNEL;
            HART_COMM_14.TimeOut := HART_TIMEOUT;

            // HART_FUNC := 'Функция 14';
            HART_FUNCTIONS := 14;

        9:  (* Функция 15 - чтение информации о выходном сигнале по первичной переменной *)
            HART_COMM_14.Request := FALSE;

            HART_COMM_15.Request := TRUE;
            HART_COMM_15.Bus := HART_BUS;
            HART_COMM_15.Device := HART_DEVICE;
            HART_COMM_15.Channel := HART_CHANNEL;
            HART_COMM_15.TimeOut := HART_TIMEOUT;

            // HART_FUNC := 'Функция 15';
            HART_FUNCTIONS := 15;

        10: (* Функция 16 - чтение сборочного номера устройства *)
            HART_COMM_15.Request := FALSE;

            HART_COMM_16.Request := TRUE;
            HART_COMM_16.Bus := HART_BUS;
            HART_COMM_16.Device := HART_DEVICE;
            HART_COMM_16.Channel := HART_CHANNEL;
            HART_COMM_16.TimeOut := HART_TIMEOUT;

            // HART_FUNC := 'Функция 16';
            HART_FUNCTIONS := 16;

        11: (* Функция 33 - чтение переменных датчика *)
            HART_COMM_16.Request := FALSE;

            HART_COMM_33.Request := TRUE;
            HART_COMM_33.Bus := HART_BUS;
            HART_COMM_33.Device := HART_DEVICE;
            HART_COMM_33.Channel := HART_CHANNEL;
            HART_COMM_33.TimeOut := HART_TIMEOUT;

            // HART_FUNC := 'Функция 33';
            HART_FUNCTIONS := 33;

        12: (* Функция 34 - запись значения демпфирования первичной переменной *)
            HART_COMM_33.Request := FALSE;

            HART_COMM_34.Request := TRUE;
            HART_COMM_34.Bus := HART_BUS;
            HART_COMM_34.Device := HART_DEVICE;
            HART_COMM_34.Channel := HART_CHANNEL;
            HART_COMM_34.TimeOut := HART_TIMEOUT;

            // HART_FUNC := 'Функция 34';
            HART_FUNCTIONS := 34;

        13: (* Функция 35 - запись значения диапазона первичной переменной *)
            HART_COMM_34.Request := FALSE;

            HART_COMM_35.Request := TRUE;
            HART_COMM_35.Bus := HART_BUS;
            HART_COMM_35.Device := HART_DEVICE;
            HART_COMM_35.Channel := HART_CHANNEL;
            HART_COMM_35.TimeOut := HART_TIMEOUT;

            // HART_FUNC := 'Функция 35';
            HART_FUNCTIONS := 35;

        14: (* Функция 48 - чтение дополнительного состояния датчика *)
            HART_COMM_35.Request := FALSE;

            HART_COMM_48.Request := TRUE;
            HART_COMM_48.Bus := HART_BUS;
            HART_COMM_48.Device := HART_DEVICE;
            HART_COMM_48.Channel := HART_CHANNEL;
            HART_COMM_48.TimeOut := HART_TIMEOUT;

            // HART_FUNC := 'Функция 48';
            HART_FUNCTIONS := 48;

        15: (* Функция 50 - чтение назначения динамических переменных *)
            HART_COMM_48.Request := FALSE;

            HART_COMM_50.Request := TRUE;
            HART_COMM_50.Bus := HART_BUS;
            HART_COMM_50.Device := HART_DEVICE;
            HART_COMM_50.Channel := HART_CHANNEL;
            HART_COMM_50.TimeOut := HART_TIMEOUT;

            // HART_FUNC := 'Функция 50';
            HART_FUNCTIONS := 50;

        16: (* Функция 54 - чтение информации о переменной датчика *)
            HART_COMM_50.Request := FALSE;

            HART_COMM_54.Request := TRUE;
            HART_COMM_54.Bus := HART_BUS;
            HART_COMM_54.Device := HART_DEVICE;
            HART_COMM_54.Channel := HART_CHANNEL;
            HART_COMM_54.TimeOut := HART_TIMEOUT;

            // HART_FUNC := 'Функция 54';
            HART_FUNCTIONS := 54;

            STEP_PULL := 0;
            FINAL_PULL := TRUE;

    END_CASE;
END_IF;

// Ошибка опроса
IF HART_COMM_00.Error <> 0
    OR HART_COMM_01.Error <> 0
    OR HART_COMM_02.Error <> 0
    OR HART_COMM_03.Error <> 0
    OR HART_COMM_06.Error <> 0
    OR HART_COMM_12.Error <> 0
    OR HART_COMM_13.Error <> 0
    OR HART_COMM_14.Error <> 0
    OR HART_COMM_15.Error <> 0
    OR HART_COMM_16.Error <> 0
    OR HART_COMM_33.Error <> 0
    OR HART_COMM_34.Error <> 0
    OR HART_COMM_35.Error <> 0
    OR HART_COMM_48.Error <> 0
    OR HART_COMM_50.Error <> 0
    OR HART_COMM_54.Error <> 0 THEN

    HART_PULL_ERROR := TRUE;

END_IF;

END_PROGRAM
